// METHODS CALLS//
	IF bInit THEN
		M_Init() ; 
		bInit	:= FALSE ; 
	ELSIF CmdInit_G  THEN 
		bInit:= TRUE ;
	END_IF
	
	M_Read();
	
	M_Evaluate();
		
	M_StateManager() ; 
	M_Write();
	M_StartStop() ; 
	

	
	M_AlarmManagement();
END_METHOD

METHOD M_Init
VAR 

END_VAR
END_METHOD

METHOD M_Read
//////////////////
//  Read Modbus Variable for racks and BBMS .  
/////////////////

VAR 
	// Method local variables (reinitialized at each cycle) 

	
END_VAR
END_METHOD

METHOD M_Write
VAR_INPUT
END_VAR
VAR
	AX_ADDR 	: ARRAY[1..1] OF UINT := [1];
	AX_QTY		: ARRAY[1..1] OF BYTE := [3];
	AX_UnitID	: ARRAY[1..1] OF BYTE := [1];
END_VAR
END_METHOD

END_FUNCTION_BLOCK

// ---- 01_Equipement_Library/Batteries/FB_SystemBMS_M3.TcPOU
FUNCTION_BLOCK FB_SystemBMS_M3 EXTENDS FB_SystemBMS_Base
// Composed of Several Racks =  A System BBMS = One DC bus independant 
// 1 Racks is composed of 1 or 2 string .  >> 1 rack = one RMBS
// 1 string is composed of several modules . >> 1 string = one DC + one DC- contactor 
// Each modules is composed of several cells . 
// 17 racks  . 

VAR_INPUT PERSISTENT
		ParamIpAddress 			: STRING 	:='192.168.1.51' ; 		// IP¨Address
		ParamUnitID				: BYTE  	:= 1 ; 					// Modbus Unit ID
		ParamTcpPort			: UINT 		:= 502;					// Modbus TCP Port
		ParamReadAlarmTime		: TIME 		:= T#90S;				// Time before communication alarm
		ParamReadWarningTime	: TIME		:= T#30S;				// Time before communication warning
		ParamClockReadRack_Delay: TIME 		:= T#500ms ; 			// Delay after bbms read and before rack read
		
		ParamNbRackString		: BYTE:=1  ; // Nb of strings of module per racks . 
		ParamNbReadAtOnce		: BYTE:=10 ; // Number of racks read at the same time . 
		
END_VAR

VAR_INPUT
	//Child objects
	
END_VAR

VAR
	
	//M_EXECUTE VARIABLES//
		AX_DFV 							: ARRAY[1..13] OF FB_DetectFixedValue;	

		
		btest							: BOOL;
END_VAR

METHOD M_Evaluate : BOOL
VAR_INPUT
END_VAR
VAR
	KK: INT;
	JJ: INT ; 
	MesUmin: REAL;
	MesUdcRack: REAL;
	CalMesCCL : REAL;
	CalMesDCL : REAL;
	CalMesIdc	: REAL;
	CalMesSoC: REAL;
	CalMesSoH: REAL;
	CalMesUdc	: REAL ; 
	CalMesUdcCell : REAL ; 
	
	CalStringsInAlarm	: INT ; 
	
	
	MesGainSoCParCycle: REAL;
	CalMesUdcConnected: REAL;
	CalMesSoCConnected: REAL;

	CalProtection: UINT;
END_VAR

// GETS COM COMMANDS , OUTPUTS  , CLOCKREAD . 


AX_TrigRead[1](CLK := ClockRead);

///// CODE EMULATION ///// 

	M_Evaluate();
	
IF AX_TrigRead[1].Q THEN
MesDataExd				:= Rea.MesDataExd.MesData.; 	
 END_IF     
 


// Initialize 
CalMesIdc := 0 ; 
CalMesCCL  := 0 ; 
CalMesDCL  := 0 ;  
CalMesSoH := 0 ; 
CalMesUdcConnected := 0 ; 
CalMesSoCConnected:= 0 ;
CalMesUdc := 0 ; 
CalMesUdcCell := 0 ;
CalStringsInAlarm := 0 ;
Rea.MesDataExd.MesData.MesRackStringState := 0 ;

// Get Data from PCS 
MesDataPcs := AX_ESS[ParamEssNum].AX_PCS[ParamSystemBmsNum].MesDataExd.MesData.
// Gestion des On et Off des DC switch
TRIG_OpenDc(CLK := CmdOpenDc);
TRIG_CloseDc(CLK := CmdCloseDc);

IF TRIG_OpenDc.Q THEN
	CmdOpenDc := FALSE;
END_IF
IF TRIG_CloseDc.Q THEN
	CmdCloseDc := FALSE;
END_IF



FOR KK := 1 TO ParamNbRacks DO
	FOR JJ:= 1 TO ParamNbRackString DO 
		
  	// check if there is a protection on either string or rack level . 
		CalProtection := Rea.MesDataExd.MesData.AX_Rack[KK].AX_RACKSTRING[JJ].MesProtection1 + Rea.MesDataExd.MesData.AX_Rack[KK].AX_RACKSTRING[JJ].MesProtection2 + Rea.MesDataExd.MesData.AX_Rack[KK].AX_RACKSTRING[JJ].MesProtection3 + Rea.MesDataExd.MesData.AX_Rack[KK].AX_RACKSTRING[JJ].MesProtection4 + Rea.MesDataExd.MesData.AX_Rack[KK].MesProtection1 + Rea.MesDataExd.MesData.AX_Rack[KK].MesProtection2  ; 
		
		IF CalProtection > 0 THEN 
			CalStringsInAlarm :=  CalStringsInAlarm + 1  ;
		END_IF
		
	TRIG_OpenDcRack[KK][JJ](CLK := Rea.MesDataExd.MesData.AX_Rack[KK].AX_RACKSTRING[JJ].MesMode = 3  AND TRIG_OpenDc.Q OR CalProtection>0);		// Opens if protection alarm
	TRIG_CloseDcRack[KK][JJ](CLK := Rea.MesDataExd.MesData.AX_Rack[KK].AX_RACKSTRING[JJ].MesMode <> 3 AND TRIG_CloseDc.Q AND CalProtection=0 );	// do not close if protection alarm
	

		IF TRIG_OpenDcRack[KK][JJ].Q THEN
			Rea.MesDataExd.MesData.AX_Rack[KK].AX_RACKSTRING[1].MesMode := 2;
			//Rea.MesDataExd.MesData.AX_Rack[KK].AX_RACKSTRING[2].MesMode := 2;	
			Rea.MesDataExd.MesData.AX_Rack[KK].MesSwitchSensorStatus := 248 ;	// protections are set and fuse are ok . Dc and ac switch are opened .
			Rea.MesDataExd.MesData.AX_Rack[KK].MesDcOpenCount			:=Rea.MesDataExd.MesData.AX_Rack[KK].MesDcOpenCount +1  ;//evaluate 
				
		END_IF
		IF TRIG_CloseDcRack[KK][JJ].Q THEN
			Rea.MesDataExd.MesData.AX_Rack[KK].AX_RACKSTRING[1].MesMode := 3;
			//Rea.MesDataExd.MesData.AX_Rack[KK].AX_RACKSTRING[2].MesMode := 3;
			Rea.MesDataExd.MesData.AX_Rack[KK].MesSwitchSensorStatus := 255 ;	// protections are set and fuse are ok . Dc and ac switch are opened .
			Rea.MesDataExd.MesData.AX_Rack[KK].MesDcCloseCount			:=Rea.MesDataExd.MesData.AX_Rack[KK].MesDcCloseCount + 1			 ;//evaluate 		
		END_IF	
	END_FOR
END_FOR

NbRacksOn := 0;

FOR KK := 1 TO ParamNbRacks DO
	FOR JJ := 1 TO ParamNbRackString DO 
		IF Rea.MesDataExd.MesData.AX_Rack[KK].AX_RACKSTRING[JJ].MesMode = 3 THEN
			NbRacksOn := NbRacksOn + 1;
		END_IF
	END_FOR
END_FOR		


FOR KK := 1 TO ParamNbRacks DO
	FOR JJ := 1 TO ParamNbRackString DO 
		IF Rea.MesDataExd.MesData.AX_Rack[KK].AX_RACKSTRING[JJ].MesMode = 3 AND NbRacksOn>=1 THEN

		Rea.MesDataExd.MesData.AX_Rack[KK].AX_RACKSTRING[JJ].MesIdc := MesDataExd.MesData.cs.CalIdc / NbRacksOn;
		MesGainSoCParCycle := Rea.MesDataExd.MesData.AX_Rack[KK].AX_RACKSTRING[JJ].MesIdc*Rea.MesDataExd.MesData.AX_Rack[KK].AX_RACKSTRING[JJ].MesUdc*(ParamCycleTime_Emul/3600000.0)/(Rea.MesDataExd.MesData.AX_Rack[KK].AX_RACKSTRING[JJ].MesSoH/100.0);
		Rea.MesDataExd.MesData.AX_Rack[KK].AX_RACKSTRING[JJ].MesSoC	 	:=MIN(MAX(0, Rea.MesDataExd.MesData.AX_Rack[KK].AX_RACKSTRING[JJ].MesSoC + MesGainSoCParCycle/CstEnergyRack*100), 100); ;//evaluate 	
		Rea.MesDataExd.MesData.AX_Rack[KK].AX_RACKSTRING[JJ].MesCCL := SEL(Rea.MesDataExd.MesData.AX_Rack[KK].AX_RACKSTRING[JJ].MesSoC < 95, (100-Rea.MesDataExd.MesData.AX_Rack[KK].AX_RACKSTRING[JJ].MesSoC)*CstEnergyRack*CstMaxCrateCharge/8000, CstEnergyRack*CstMaxCrateCharge*CstNominalVoltage/Rea.MesDataExd.MesData.AX_Rack[KK].AX_RACKSTRING[JJ].MesUdc_Cell/1000);
		Rea.MesDataExd.MesData.AX_Rack[KK].AX_RACKSTRING[JJ].MesDCL := SEL(Rea.MesDataExd.MesData.AX_Rack[KK].AX_RACKSTRING[JJ].MesSoC > 5, Rea.MesDataExd.MesData.AX_Rack[KK].AX_RACKSTRING[JJ].MesSoC*CstEnergyRack*CstMaxCrateDischarge/8000, CstEnergyRack*CstMaxCrateDischarge*CstNominalVoltage/Rea.MesDataExd.MesData.AX_Rack[KK].AX_RACKSTRING[JJ].MesUdc_Cell/1000);
		Rea.MesDataExd.MesData.AX_Rack[KK].AX_RACKSTRING[JJ].MesState.1 := SEL(Rea.MesDataExd.MesData.AX_Rack[KK].AX_RACKSTRING[JJ].MesIdc <> 0 , TRUE  , FALSE )  ; 
		CalMesUdcConnected := CalMesUdcConnected + Rea.MesDataExd.MesData.AX_Rack[KK].AX_RACKSTRING[JJ].MesUdc / NbRacksOn ; 
		CalMesSoCConnected := CalMesSoCConnected  +  Rea.MesDataExd.MesData.AX_Rack[KK].AX_RACKSTRING[JJ].MesSoC / NbRacksOn ; 
		ELSE
			Rea.MesDataExd.MesData.AX_Rack[KK].AX_RACKSTRING[JJ].MesIdc := 0;
			Rea.MesDataExd.MesData.AX_Rack[KK].AX_RACKSTRING[JJ].MesCCL := 0;
			Rea.MesDataExd.MesData.AX_Rack[KK].AX_RACKSTRING[JJ].MesDCL :=0;
			Rea.MesDataExd.MesData.AX_Rack[KK].AX_RACKSTRING[JJ].MesState := 0  ; 	
		END_IF
		
		MesUmin := ParamUdcMin +(ParamUdcMax - ParamUdcMin) * Rea.MesDataExd.MesData.AX_Rack[KK].AX_RACKSTRING[JJ].MesSoC /100;
		Rea.MesDataExd.MesData.AX_Rack[KK].AX_RACKSTRING[JJ].MesUdc			:=MesUmin ;//evaluate 
		Rea.MesDataExd.MesData.AX_Rack[KK].AX_RACKSTRING[JJ].MesUdc_ModuleSum	:=MesUmin ;//evaluate 		
		Rea.MesDataExd.MesData.AX_Rack[KK].AX_RACKSTRING[JJ].MesUdc_CellSum	:=MesUmin ;//evaluate 			
		Rea.MesDataExd.MesData.AX_Rack[KK].AX_RACKSTRING[JJ].MesIdc_Avg		:=Rea.MesDataExd.MesData.AX_Rack[KK].AX_RACKSTRING[JJ].MesIdc ;//evaluate 		
			
		Rea.MesDataExd.MesData.AX_Rack[KK].AX_RACKSTRING[JJ].MesCPL		:=Rea.MesDataExd.MesData.AX_Rack[KK].AX_RACKSTRING[JJ].MesCCL * Rea.MesDataExd.MesData.AX_Rack[KK].AX_RACKSTRING[JJ].MesUdc ;//evaluate 	
		Rea.MesDataExd.MesData.AX_Rack[KK].AX_RACKSTRING[JJ].MesDPL		:=Rea.MesDataExd.MesData.AX_Rack[KK].AX_RACKSTRING[JJ].MesDCL * Rea.MesDataExd.MesData.AX_Rack[KK].AX_RACKSTRING[JJ].MesUdc ;//evaluate 

		IF Rea.MesDataExd.MesData.AX_Rack[KK].AX_RACKSTRING[JJ].MesIdc > 0 THEN 
			Rea.MesDataExd.MesData.AX_Rack[KK].AX_RACKSTRING[JJ].MesECharge := Rea.MesDataExd.MesData.AX_Rack[KK].AX_RACKSTRING[JJ].MesECharge + Rea.MesDataExd.MesData.AX_Rack[KK].AX_RACKSTRING[JJ].MesIdc*Rea.MesDataExd.MesData.AX_Rack[KK].AX_RACKSTRING[JJ].MesUdc*ParamCycleTime_Emul/3600000.0 ;
		ELSE 
			Rea.MesDataExd.MesData.AX_Rack[KK].AX_RACKSTRING[JJ].MesEDischarge := Rea.MesDataExd.MesData.AX_Rack[KK].AX_RACKSTRING[JJ].MesEDischarge - Rea.MesDataExd.MesData.AX_Rack[KK].AX_RACKSTRING[JJ].MesIdc*Rea.MesDataExd.MesData.AX_Rack[KK].AX_RACKSTRING[JJ].MesUdc*ParamCycleTime_Emul/3600000.0 ;

		END_IF

		Rea.MesDataExd.MesData.AX_Rack[KK].AX_RACKSTRING[JJ].MesUdc_Cell		:=Rea.MesDataExd.MesData.AX_Rack[KK].AX_RACKSTRING[JJ].MesUdc / 264 ;//evaluate Nb of cells per strings 
		Rea.MesDataExd.MesData.AX_Rack[KK].AX_RACKSTRING[JJ].MesUdcMax1_Cell	:=Rea.MesDataExd.MesData.AX_Rack[KK].AX_RACKSTRING[JJ].MesUdc_Cell ;//evaluate 
		Rea.MesDataExd.MesData.AX_Rack[KK].AX_RACKSTRING[JJ].MesUdcMin1_Cell:=Rea.MesDataExd.MesData.AX_Rack[KK].AX_RACKSTRING[JJ].MesUdc_Cell ;//evaluate 
		Rea.MesDataExd.MesData.AX_Rack[KK].AX_RACKSTRING[JJ].MesUdcMax2_Cell	:=Rea.MesDataExd.MesData.AX_Rack[KK].AX_RACKSTRING[JJ].MesUdc_Cell ;//evaluate 
		Rea.MesDataExd.MesData.AX_Rack[KK].AX_RACKSTRING[JJ].MesUdcMin2_Cell:=Rea.MesDataExd.MesData.AX_Rack[KK].AX_RACKSTRING[JJ].MesUdc_Cell ;//evaluate 
		
		Rea.MesDataExd.MesData.MesRackStringState			        := Rea.MesDataExd.MesData.MesRackStringState OR Rea.MesDataExd.MesData.AX_Rack[KK].AX_RACKSTRING[JJ].MesState;//evaluate 
				
		CalMesIdc := CalMesIdc +  Rea.MesDataExd.MesData.AX_Rack[KK].AX_RACKSTRING[JJ].MesIdc ;
		CalMesCCL  	:= CalMesCCL + Rea.MesDataExd.MesData.AX_Rack[KK].Ax_RACKSTRING[JJ].MesCCL; 
		CalMesDCL  	:= CalMesDCL + Rea.MesDataExd.MesData.AX_Rack[KK].Ax_RACKSTRING[JJ].MesDCL; 
		CalMesSoC 	:= CalMesSoC + Rea.MesDataExd.MesData.AX_Rack[KK].Ax_RACKSTRING[JJ].MesSoC / ParamNbRacks; 
		CalMesUdc := CalMesUdc + Rea.MesDataExd.MesData.AX_Rack[KK].AX_RACKSTRING[JJ].MesUdc / ParamNbRacks ; 
		CalMesUdcCell := CalMesUdcCell  + Rea.MesDataExd.MesData.AX_Rack[KK].AX_RACKSTRING[JJ].MesUdc_Cell / ParamNbRacks ;

	END_FOR

	Rea.MesDataExd.MesData.AX_Rack[KK].MesHeartBeat		:=WORD_TO_UINT(CalLocalTimeStruct.wSecond); ;//evaluate 

END_FOR	

Rea.MesDataExd.MesData.MesHeartBeat						:=WORD_TO_UINT(CalLocalTimeStruct.wSecond); ;//evaluate			
Rea.MesDataExd.MesData.MesNbRackConnected			        :=NbRacksOn ;//evaluate
Rea.MesDataExd.MesData.MesIdcConnected				        :=CalMesIdc ;//evaluate
Rea.MesDataExd.MesData.MesUdcConnected				        :=CalMesUdcConnected ;//evaluate
Rea.MesDataExd.MesData.MesUdcConnectedMedian		        :=CalMesUdcConnected ;//evaluate
Rea.MesDataExd.MesData.MesUdcConnectedMax			        := CalMesUdcConnected;//evaluate
Rea.MesDataExd.MesData.MesUdcConnectedMin			        := CalMesUdcConnected;//evaluate
Rea.MesDataExd.MesData.MesSoCConnected				        := CalMesSoCConnected;//evaluate average 
Rea.MesDataExd.MesData.MesSoCConnectedMedian		        := CalMesSoCConnected;//evaluate
Rea.MesDataExd.MesData.MesSoCConnectedMax			        := CalMesSoCConnected;//evaluate
Rea.MesDataExd.MesData.MesSoCConnectedMin			        := CalMesSoCConnected;//evaluate
Rea.MesDataExd.MesData.MesIdc						        := CalMesIdc;//evaluate
Rea.MesDataExd.MesData.MesUdc						        := CalMesUdc;//evaluate
Rea.MesDataExd.MesData.MesUdcMedian				        := CalMesUdc;//evaluate
Rea.MesDataExd.MesData.MesUdcMax					        := CalMesUdc;//evaluate
Rea.MesDataExd.MesData.MesUdcMin					        := CalMesUdc;//evaluate
Rea.MesDataExd.MesData.MesSoC						        := CalMesSoC;//evaluate
Rea.MesDataExd.MesData.MesSoCMedian				        := CalMesSoC;//evaluate
Rea.MesDataExd.MesData.MesSoCMax					        := CalMesSoC;//evaluate
Rea.MesDataExd.MesData.MesSoCMin					        := CalMesSoC;//evaluate
Rea.MesDataExd.MesData.MesUdc_Cell					        := CalMesUdcCell;//evaluate
Rea.MesDataExd.MesData.MesUdcMedian_Cell			        := CalMesUdcCell;//evaluate
Rea.MesDataExd.MesData.MesUdcMax_Cell				        := CalMesUdcCell;//evaluate
Rea.MesDataExd.MesData.MesUdcMin_Cell				        := CalMesUdcCell;//evaluate
Rea.MesDataExd.MesData.MesCCL						        := CalMesCCL;//evaluate
Rea.MesDataExd.MesData.MesDCL						        := CalMesDCL;//evaluate
Rea.MesDataExd.MesData.MesCPL						        := CalMesCCL *Rea.MesDataExd.MesData.MesUdc ;//evaluate
Rea.MesDataExd.MesData.MesDPL						        := CalMesDCL *Rea.MesDataExd.MesData.MesUdc;//evaluate
IF Rea.MesDataExd.MesData.MesIdc > 0 THEN 
	Rea.MesDataExd.MesData.MesECharge := Rea.MesDataExd.MesData.MesECharge + Rea.MesDataExd.MesData.MesIdc*Rea.MesDataExd.MesData.MesUdc*ParamCycleTime_Emul/3600000.0 ;
ELSE 
	Rea.MesDataExd.MesData.MesEDischarge := Rea.MesDataExd.MesData.MesEDischarge - Rea.MesDataExd.MesData.MesIdc*Rea.MesDataExd.MesData.MesUdc*ParamCycleTime_Emul/3600000.0 ;

END_IF

Rea.MesDataExd.MesData.MesWatchdog					        := AX_Cmd[3];//evaluate

Rea.MesDataExd.MesData.MesSystemMode.15				     := Rea.MesDataExd.MesData.MesIdc < - (3 * Rea.MesDataExd.MesData.MesNbRackConnected) ;//discharge 
Rea.MesDataExd.MesData.MesSystemMode.14				     := Rea.MesDataExd.MesData.MesIdc > 3  *Rea.MesDataExd.MesData.MesNbRackConnected ;//discharge 




Rea.MesDataExd.MesData.MesSystemMode.2:= SEL(CalStringsInAlarm = 0 AND Rea.MesDataExd.MesData.MesNbRackConnected =0  , FALSE ,  TRUE )  ;		// all strings can be connected 
Rea.MesDataExd.MesData.MesSystemMode.3:= NOT Rea.MesDataExd.MesData.MesSystemMode.2 AND SEL(CalStringsInAlarm < ( Rea.MesDataExd.MesData.MesNbRackTot - Rea.MesDataExd.MesData.ParamStringNbMin ) AND Rea.MesDataExd.MesData.MesNbRackConnected =0  , FALSE ,  TRUE )  ;		// Part of strings can be connected 
Rea.MesDataExd.MesData.MesSystemMode.4:= SEL(CalStringsInAlarm >= ( Rea.MesDataExd.MesData.MesNbRackTot - Rea.MesDataExd.MesData.ParamStringNbMin ) AND Rea.MesDataExd.MesData.MesNbRackConnected =0 , FALSE ,  TRUE )  ;	// 
Rea.MesDataExd.MesData.MesSystemMode.5:= SEL(CalStringsInAlarm = 0 AND Rea.MesDataExd.MesData.MesNbRackConnected >0  , FALSE ,  TRUE )  ;
Rea.MesDataExd.MesData.MesSystemMode.6:= NOT Rea.MesDataExd.MesData.MesSystemMode.5 AND SEL(CalStringsInAlarm > 0 AND Rea.MesDataExd.MesData.MesNbRackConnected =0  , FALSE ,  TRUE )  ;
END_METHOD

METHOD M_Init
VAR 
KK:  INT  ; 

	JJ: INT;
END_VAR
FOR KK := 1 TO ParamNbRacks DO
	FOR JJ := 1 TO ParamNbRackString DO 
		Rea.MesDataExd.MesData.AX_Rack[KK].AX_RACKSTRING[JJ].MesMode						:=2  ;//evaluate 				
		Rea.MesDataExd.MesData.AX_Rack[KK].AX_RACKSTRING[JJ].MesAlarm1					    :=0  ;//init 
		Rea.MesDataExd.MesData.AX_Rack[KK].AX_RACKSTRING[JJ].MesAlarm2						:=0  ;//init  	
		Rea.MesDataExd.MesData.AX_Rack[KK].AX_RACKSTRING[JJ].MesAlarm3						:=0  ;//init  	
		Rea.MesDataExd.MesData.AX_Rack[KK].AX_RACKSTRING[JJ].MesAlarm4						:=0  ;//init  	
		Rea.MesDataExd.MesData.AX_Rack[KK].AX_RACKSTRING[JJ].MesProtection1				:=0  ;//init  		
		Rea.MesDataExd.MesData.AX_Rack[KK].AX_RACKSTRING[JJ].MesProtection2				:=0  ;//init  		
		Rea.MesDataExd.MesData.AX_Rack[KK].AX_RACKSTRING[JJ].MesProtection3				:=0  ;//init  		
		Rea.MesDataExd.MesData.AX_Rack[KK].AX_RACKSTRING[JJ].MesProtection4				:=0  ;//init  		
		Rea.MesDataExd.MesData.AX_Rack[KK].AX_RACKSTRING[JJ].MesControlStatus				:=1  ;//init  	
		Rea.MesDataExd.MesData.AX_Rack[KK].AX_RACKSTRING[JJ].MesUdc						:=850  ;//evaluate 		
		Rea.MesDataExd.MesData.AX_Rack[KK].AX_RACKSTRING[JJ].MesUdc_ModuleSum				:=850  ;//evaluate	
		Rea.MesDataExd.MesData.AX_Rack[KK].AX_RACKSTRING[JJ].MesUdc_CellSum				:=850  ;//evaluate
		Rea.MesDataExd.MesData.AX_Rack[KK].AX_RACKSTRING[JJ].MesIdc						:=0  ;//evaluate	
		Rea.MesDataExd.MesData.AX_Rack[KK].AX_RACKSTRING[JJ].MesIdc_Avg					:=0  ;//evaluate	
		Rea.MesDataExd.MesData.AX_Rack[KK].AX_RACKSTRING[JJ].MesSoC	 					:=50  ;//evaluate	
		Rea.MesDataExd.MesData.AX_Rack[KK].AX_RACKSTRING[JJ].MesSoH	 					:=100  ;//evaluate	
		Rea.MesDataExd.MesData.AX_Rack[KK].AX_RACKSTRING[JJ].MesCCL						:=0  ;//evaluate	
		Rea.MesDataExd.MesData.AX_Rack[KK].AX_RACKSTRING[JJ].MesDCL						:=0  ;//evaluate	
		Rea.MesDataExd.MesData.AX_Rack[KK].AX_RACKSTRING[JJ].MesCPL						:=0  ;//evaluate	
		Rea.MesDataExd.MesData.AX_Rack[KK].AX_RACKSTRING[JJ].MesDPL						:=0  ;//evaluate	
		Rea.MesDataExd.MesData.AX_Rack[KK].AX_RACKSTRING[JJ].MesECharge					:=0  ;//evaluate	
		Rea.MesDataExd.MesData.AX_Rack[KK].AX_RACKSTRING[JJ].MesEDischarge					:=0  ;//evaluate
		Rea.MesDataExd.MesData.AX_Rack[KK].AX_RACKSTRING[JJ].MesOff_ModuleID				:=1  ;//init 		
		Rea.MesDataExd.MesData.AX_Rack[KK].AX_RACKSTRING[JJ].MesComError_ModuleID			:=1  ;//init 	
		Rea.MesDataExd.MesData.AX_Rack[KK].AX_RACKSTRING[JJ].MesUdcDiffMax_Cell			:=0  ;//init 		
		Rea.MesDataExd.MesData.AX_Rack[KK].AX_RACKSTRING[JJ].MesUdc_Cell					:=30  ;//evaluate		
		Rea.MesDataExd.MesData.AX_Rack[KK].AX_RACKSTRING[JJ].MesUdcMax1_Cell				:=30  ;//evaluate		
		Rea.MesDataExd.MesData.AX_Rack[KK].AX_RACKSTRING[JJ].MesUdcMax1_Cell_ModuleID		:=1  ;//init 	
		Rea.MesDataExd.MesData.AX_Rack[KK].AX_RACKSTRING[JJ].MesUdcMax1_Cell_CellID		:=1  ;//init 		
		Rea.MesDataExd.MesData.AX_Rack[KK].AX_RACKSTRING[JJ].MesUdcMin1_Cell				:=30  ;//evaluate		
		Rea.MesDataExd.MesData.AX_Rack[KK].AX_RACKSTRING[JJ].MesUdcMin1_Cell_ModuleID		:=1  ;//init 	
		Rea.MesDataExd.MesData.AX_Rack[KK].AX_RACKSTRING[JJ].MesUdcMin1_Cell_CellID		:=1  ;//init 		
		Rea.MesDataExd.MesData.AX_Rack[KK].AX_RACKSTRING[JJ].MesUdcMax2_Cell				:=30  ;//evaluate		
		Rea.MesDataExd.MesData.AX_Rack[KK].AX_RACKSTRING[JJ].MesUdcMax2_Cell_ModuleID		:=1  ;//init 	
		Rea.MesDataExd.MesData.AX_Rack[KK].AX_RACKSTRING[JJ].MesUdcMax2_Cell_CellID		:=1  ;//init 		
		Rea.MesDataExd.MesData.AX_Rack[KK].AX_RACKSTRING[JJ].MesUdcMin2_Cell				:=30  ;//evaluate		
		Rea.MesDataExd.MesData.AX_Rack[KK].AX_RACKSTRING[JJ].MesUdcMin2_Cell_ModuleID		:= 1 ;//init 	
		Rea.MesDataExd.MesData.AX_Rack[KK].AX_RACKSTRING[JJ].MesUdcMin2_Cell_CellID		:= 1 ;//init 		
		Rea.MesDataExd.MesData.AX_Rack[KK].AX_RACKSTRING[JJ].MesTempDiffMax_Cell			:=0  ;//init		
		Rea.MesDataExd.MesData.AX_Rack[KK].AX_RACKSTRING[JJ].MesTemp_Cell					:=25  ;// init	
		Rea.MesDataExd.MesData.AX_Rack[KK].AX_RACKSTRING[JJ].MesTempMax1_Cell				:=25  ;//init 	
		Rea.MesDataExd.MesData.AX_Rack[KK].AX_RACKSTRING[JJ].MesTempMax1_Cell_ModuleID		:=4  ;//init 	
		Rea.MesDataExd.MesData.AX_Rack[KK].AX_RACKSTRING[JJ].MesTempMax1_Cell_CellID		:=4  ;//init 		
		Rea.MesDataExd.MesData.AX_Rack[KK].AX_RACKSTRING[JJ].MesTempMin1_Cell				:=20  ;//init 	
		Rea.MesDataExd.MesData.AX_Rack[KK].AX_RACKSTRING[JJ].MesTempMin1_Cell_ModuleID		:= 1 ;//init 	
		Rea.MesDataExd.MesData.AX_Rack[KK].AX_RACKSTRING[JJ].MesTempMin1_Cell_CellID		:= 1 ;//init 		
		Rea.MesDataExd.MesData.AX_Rack[KK].AX_RACKSTRING[JJ].MesTempMax2_Cell				:=23  ;//init 	
		Rea.MesDataExd.MesData.AX_Rack[KK].AX_RACKSTRING[JJ].MesTempMax2_Cell_ModuleID		:=3  ;//init 	
		Rea.MesDataExd.MesData.AX_Rack[KK].AX_RACKSTRING[JJ].MesTempMax2_Cell_CellID		:=3  ;//init 		
		Rea.MesDataExd.MesData.AX_Rack[KK].AX_RACKSTRING[JJ].MesTempMin2_Cell				:=21  ;//init 	
		Rea.MesDataExd.MesData.AX_Rack[KK].AX_RACKSTRING[JJ].MesTempMin2_Cell_ModuleID		:=2  ;//init 	
		Rea.MesDataExd.MesData.AX_Rack[KK].AX_RACKSTRING[JJ].MesTempMin2_Cell_CellID		:=2  ;//init 		
		Rea.MesDataExd.MesData.AX_Rack[KK].AX_RACKSTRING[JJ].MesTempPCBMax					:=31  ;//init 	
		Rea.MesDataExd.MesData.AX_Rack[KK].AX_RACKSTRING[JJ].MesTempPCBMax_ModuleID		:=5  ;//init 		
		Rea.MesDataExd.MesData.AX_Rack[KK].AX_RACKSTRING[JJ].MesTempPCBMin					:=28  ;//init 	
		Rea.MesDataExd.MesData.AX_Rack[KK].AX_RACKSTRING[JJ].MesTempPCBMin_ModuleID		:=6  ;//init 		
		Rea.MesDataExd.MesData.AX_Rack[KK].AX_RACKSTRING[JJ].MesSensorStatus				:=0  ;//init 		
		Rea.MesDataExd.MesData.AX_Rack[KK].AX_RACKSTRING[JJ].MesModuleScanStatus			:=0  ;//init 		
		Rea.MesDataExd.MesData.AX_Rack[KK].AX_RACKSTRING[JJ].MesModuleBalancingStatus		:=0  ;//init 	
		Rea.MesDataExd.MesData.AX_Rack[KK].AX_RACKSTRING[JJ].MesModuleAddressStatus		:=0  ;//init 		
		Rea.MesDataExd.MesData.AX_Rack[KK].AX_RACKSTRING[JJ].MesModuleVoltageStatus		:=0  ;//init 		
		Rea.MesDataExd.MesData.AX_Rack[KK].AX_RACKSTRING[JJ].MesModuleTemperatureStatus	:=0  ;//init 		
		Rea.MesDataExd.MesData.AX_Rack[KK].AX_RACKSTRING[JJ].MesState						:=0  ;//evaluate	
		
	END_FOR
	Rea.MesDataExd.MesData.AX_Rack[KK].ParamNbStrings			:=1 ; //init 	
	Rea.MesDataExd.MesData.AX_Rack[KK].MesHeartBeat			:= 1;//evaluate 	
	Rea.MesDataExd.MesData.AX_Rack[KK].MesAlarm1				:=0 ;//init  	
	Rea.MesDataExd.MesData.AX_Rack[KK].MesAlarm2				:=0 ;//init  	
	Rea.MesDataExd.MesData.AX_Rack[KK].MesProtection1			:=0 ;//init  	
	Rea.MesDataExd.MesData.AX_Rack[KK].MesProtection2			:=0 ;//init  	
	Rea.MesDataExd.MesData.AX_Rack[KK].MesSwitchControlStatus	:=0 ;//init  	
	Rea.MesDataExd.MesData.AX_Rack[KK].MesSwitchSensorStatus	:=0 ;//evaluate  	
	Rea.MesDataExd.MesData.AX_Rack[KK].MesUSwtchGrPackPlus		:=48 ;//init  	
	Rea.MesDataExd.MesData.AX_Rack[KK].MesTempPCB				:=25.5 ;//init  
	Rea.MesDataExd.MesData.AX_Rack[KK].MesIdcFaultLvl			:=79 ;//init  
	Rea.MesDataExd.MesData.AX_Rack[KK].MesDcOpenCount			:=0 ;//evaluate 
	Rea.MesDataExd.MesData.AX_Rack[KK].MesDcCloseCount			:=0 ;//evaluate 
	
		
END_FOR	
Rea.MesDataExd.MesData.MesHeartBeat						:=1 ;//evaluate			
Rea.MesDataExd.MesData.MesNbRackConnected			        :=17 ;//evaluate
Rea.MesDataExd.MesData.MesNbRackTot				        :=17 ;//evaluate 
Rea.MesDataExd.MesData.MesIdcConnected				        :=0 ;//evaluate
Rea.MesDataExd.MesData.MesUdcConnected				        :=850 ;//evaluate
Rea.MesDataExd.MesData.MesUdcConnectedMedian		        :=850 ;//evaluate
Rea.MesDataExd.MesData.MesUdcConnectedMax			        := 850;//evaluate
Rea.MesDataExd.MesData.MesUdcConnectedMin			        := 850;//evaluate
Rea.MesDataExd.MesData.MesSoCConnected				        := 50;//evaluate
Rea.MesDataExd.MesData.MesSoCConnectedMedian		        := 50;//evaluate
Rea.MesDataExd.MesData.MesSoCConnectedMax			        := 50;//evaluate
Rea.MesDataExd.MesData.MesSoCConnectedMin			        := 50;//evaluate
Rea.MesDataExd.MesData.MesIdc						        := 0;//evaluate
Rea.MesDataExd.MesData.MesUdc						        := 850;//evaluate
Rea.MesDataExd.MesData.MesUdcMedian				        := 850;//evaluate
Rea.MesDataExd.MesData.MesUdcMax					        := 850;//evaluate
Rea.MesDataExd.MesData.MesUdcMin					        := 850;//evaluate
Rea.MesDataExd.MesData.MesSoC						        := 50;//evaluate
Rea.MesDataExd.MesData.MesSoCMedian				        := 50;//evaluate
Rea.MesDataExd.MesData.MesSoCMax					        := 50;//evaluate
Rea.MesDataExd.MesData.MesSoCMin					        := 50;//evaluate
Rea.MesDataExd.MesData.MesSoH						        := 100;//init
Rea.MesDataExd.MesData.MesSoHMedian				        := 100;//init 
Rea.MesDataExd.MesData.MesSoHMax					        := 100;//init 
Rea.MesDataExd.MesData.MesSoHMin					        := 100;//init 
Rea.MesDataExd.MesData.MesUdc_Cell					        := 30;//evaluate
Rea.MesDataExd.MesData.MesUdcMedian_Cell			        := 30;//evaluate
Rea.MesDataExd.MesData.MesUdcMax_Cell				        := 30;//evaluate
Rea.MesDataExd.MesData.MesUdcMax_Cell_RackID		        := 30;//init 
Rea.MesDataExd.MesData.MesUdcMin_Cell				        := 30;//evaluate
Rea.MesDataExd.MesData.MesUdcMin_Cell_RackID		        := 1;//init 
Rea.MesDataExd.MesData.MesUdcDiffMax_Cell			        :=0 ;//init
Rea.MesDataExd.MesData.MesUdcDiffMax_Cell_RackID	        := 1;//init 
Rea.MesDataExd.MesData.MesTmp_Cell					        := 25;//init 
Rea.MesDataExd.MesData.MesTmpMedian_Cell			        := 25;//init 
Rea.MesDataExd.MesData.MesTmpMax_Cell				        := 25;//init 
Rea.MesDataExd.MesData.MesTmpMax_Cell_RackID		        := 3;//init 
Rea.MesDataExd.MesData.MesTmpMin_Cell				        := 25;//init 
Rea.MesDataExd.MesData.MesTmpMin_Cell_RackID		        := 4;//init 
Rea.MesDataExd.MesData.MesTmpDiffMax_Cell			        := 0;//init 
Rea.MesDataExd.MesData.MesTmpDiffMax_Cell_RackID	        := 3;//init 
Rea.MesDataExd.MesData.MesCCL						        := 0;//evaluate
Rea.MesDataExd.MesData.MesDCL						        := 0;//evaluate
Rea.MesDataExd.MesData.MesCPL						        := 0;//evaluate
Rea.MesDataExd.MesData.MesDPL						        := 0;//evaluate
Rea.MesDataExd.MesData.MesECharge					        := 0;//evaluate
Rea.MesDataExd.MesData.MesEDischarge				        := 0;//evaluate
Rea.MesDataExd.MesData.MesWatchdog					        := 0;//evaluate
Rea.MesDataExd.MesData.MesUdc_PartialOp			        := 850;//evaluate
Rea.MesDataExd.MesData.MesUdc_PartialOp_RackID		        := 8;//init 
Rea.MesDataExd.MesData.MesUdc_PartialOp_StringID	        := 3;//init 
Rea.MesDataExd.MesData.MesSystemCommandStatus		        := 0;//init 
Rea.MesDataExd.MesData.MesSystemMode				        := 0;//evaluate 
Rea.MesDataExd.MesData.MesSystemMode2				        := 0;//evaluate 
Rea.MesDataExd.MesData.MesAlarm1					        := 0;//init 
Rea.MesDataExd.MesData.MesAlarm2					        := 0;//init 
Rea.MesDataExd.MesData.MesRackAlarm1				        := 0;//init
Rea.MesDataExd.MesData.MesRackAlarm2				        := 0;//init
Rea.MesDataExd.MesData.MesRackProtection1			        := 0;//init
Rea.MesDataExd.MesData.MesRackProtection2			        := 0;//init
Rea.MesDataExd.MesData.MesRackStringAlarm1			        := 0;//init
Rea.MesDataExd.MesData.MesRackStringAlarm2			        := 0;//init
Rea.MesDataExd.MesData.MesRackStringAlarm3			        := 0;//init
Rea.MesDataExd.MesData.MesRackStringAlarm4			        := 0;//init
Rea.MesDataExd.MesData.MesRackStringProtection1	        := 0;//init
Rea.MesDataExd.MesData.MesRackStringProtection2	        := 0;//init
Rea.MesDataExd.MesData.MesRackStringProtection3	        := 0;//init
Rea.MesDataExd.MesData.MesRackStringProtection4	        := 0;//init
Rea.MesDataExd.MesData.MesDiStatus					        := 0;//init
Rea.MesDataExd.MesData.MesDoStatus					        := 0;//init
Rea.MesDataExd.MesData.MesSystemConfig1			        := 0;//init
Rea.MesDataExd.MesData.MesSystemConfig2			        := 0;//init
Rea.MesDataExd.MesData.MesRackStringState			        := 0;//evaluate 
Rea.MesDataExd.MesData.ParamNbRacks				        := 17;//init
Rea.MesDataExd.MesData.ParamNbModule				        := 25;//init
Rea.MesDataExd.MesData.ParamStringNbMin			        := 10;//init
Rea.MesDataExd.MesData.ParamUdiff					        := 5;//init


SUPER^.M_Init() ;
END_METHOD

METHOD M_Read
//////////////////
//  Read CAN 2.0B Variables for racks and BBMS .  
/////////////////

VAR 
	// Method local variables (reinitialized at each cycle) 
	MW 	: FB_MergeWordsToDint ; 

	AX_Addr		: ARRAY[1..2] OF UINT := [16#00	,  16#3E8];
	AX_Qty		: ARRAY[1..3] OF UINT := [	112		, 35	,97	];
	LL			: INT;
	KK			: BYTE;
	CalRackNb	: INT;
	JJ			: BYTE;

END_VAR
// System BMS 
IF MesCP_Read  THEN	

	ModbusRead
	(
		pDestAddr 		:= ADR(MesBlock1_Temp),		sIPAddr 		:= ParamIpAddress,			tTimeout 		:= ParamTimeout,
		nTcpPort 		:= ParamTcpPort,				nQuantity 		:= AX_Qty[1],				nMBAddr 		:= AX_Addr[1],				
		cbLength 		:= SIZEOF(MesBlock1_Temp),	nUnitID 		:= ParamUnitID,				ClockRead 		:= Clockread AND  MesCP_Read,
		Reset 			:= IN_CmdReset_L,					ModbusReadAlarm => MesModbusReadAlarm,	ErrorId 		=> MesModbusReadAlarmID
	);



MesDataExd.MesData.MesHeartBeat:=MesBlock1_Temp[0];
MesDataExd.MesData.MesNbRackConnected:=MesBlock1_Temp[1];
MesDataExd.MesData.MesNbRackTot:=MesBlock1_Temp[2];
	MW(WORD_STRONG:= MesBlock1_Temp[ 3], SIGNED:=TRUE, FIX:=0 , SIZE:=1, VAR_OUT := MesDataExd.MesData.MesIdcConnected);
	MW(WORD_STRONG:= MesBlock1_Temp[ 4], SIGNED:=FALSE, FIX:=1 , SIZE:=1, VAR_OUT := MesDataExd.MesData.MesUdcConnected);
	MW(WORD_STRONG:= MesBlock1_Temp[ 5], SIGNED:=FALSE, FIX:=1 , SIZE:=1, VAR_OUT := MesDataExd.MesData.MesUdcConnectedMedian);
	MW(WORD_STRONG:= MesBlock1_Temp[ 6], SIGNED:=FALSE, FIX:=1 , SIZE:=1, VAR_OUT := MesDataExd.MesData.MesUdcConnectedMax);
	MW(WORD_STRONG:= MesBlock1_Temp[ 7], SIGNED:=FALSE, FIX:=1 , SIZE:=1, VAR_OUT := MesDataExd.MesData.MesUdcConnectedMin);
	MW(WORD_STRONG:= MesBlock1_Temp[ 8], SIGNED:=FALSE, FIX:=1 , SIZE:=1, VAR_OUT := MesDataExd.MesData.MesSoCConnected);
	MW(WORD_STRONG:= MesBlock1_Temp[ 9], SIGNED:=FALSE, FIX:=1 , SIZE:=1, VAR_OUT := MesDataExd.MesData.MesSoCConnectedMedian);
	MW(WORD_STRONG:= MesBlock1_Temp[ 10], SIGNED:=FALSE, FIX:=1 , SIZE:=1, VAR_OUT := MesDataExd.MesData.MesSoCConnectedMax);
	MW(WORD_STRONG:= MesBlock1_Temp[ 11], SIGNED:=FALSE, FIX:=1 , SIZE:=1, VAR_OUT := MesDataExd.MesData.MesSoCConnectedMin);
	MW(WORD_STRONG:= MesBlock1_Temp[ 12], SIGNED:=TRUE, FIX:=0 , SIZE:=1, VAR_OUT := MesDataExd.MesData.MesIdc);
	MW(WORD_STRONG:= MesBlock1_Temp[ 13], SIGNED:=FALSE, FIX:=1 , SIZE:=1, VAR_OUT := MesDataExd.MesData.MesUdc);
	MW(WORD_STRONG:= MesBlock1_Temp[ 14], SIGNED:=FALSE, FIX:=1 , SIZE:=1, VAR_OUT := MesDataExd.MesData.MesUdcMedian);
	MW(WORD_STRONG:= MesBlock1_Temp[ 15], SIGNED:=FALSE, FIX:=1 , SIZE:=1, VAR_OUT := MesDataExd.MesData.MesUdcMax);
	MW(WORD_STRONG:= MesBlock1_Temp[ 16], SIGNED:=FALSE, FIX:=1 , SIZE:=1, VAR_OUT := MesDataExd.MesData.MesUdcMin);
	MW(WORD_STRONG:= MesBlock1_Temp[ 17], SIGNED:=FALSE, FIX:=1 , SIZE:=1, VAR_OUT := MesDataExd.MesData.MesSoC);
	MW(WORD_STRONG:= MesBlock1_Temp[ 18], SIGNED:=FALSE, FIX:=1 , SIZE:=1, VAR_OUT := MesDataExd.MesData.MesSoCMedian);
	MW(WORD_STRONG:= MesBlock1_Temp[ 19], SIGNED:=FALSE, FIX:=1 , SIZE:=1, VAR_OUT := MesDataExd.MesData.MesSoCMax);
	MW(WORD_STRONG:= MesBlock1_Temp[ 20], SIGNED:=FALSE, FIX:=1 , SIZE:=1, VAR_OUT := MesDataExd.MesData.MesSoCMin);
	MW(WORD_STRONG:= MesBlock1_Temp[ 21], SIGNED:=FALSE, FIX:=1 , SIZE:=1, VAR_OUT := MesDataExd.MesData.MesSoH);
	MW(WORD_STRONG:= MesBlock1_Temp[ 22], SIGNED:=FALSE, FIX:=1 , SIZE:=1, VAR_OUT := MesDataExd.MesData.MesSoHMedian);
	MW(WORD_STRONG:= MesBlock1_Temp[ 23], SIGNED:=FALSE, FIX:=1 , SIZE:=1, VAR_OUT := MesDataExd.MesData.MesSoHMax);
	MW(WORD_STRONG:= MesBlock1_Temp[ 24], SIGNED:=FALSE, FIX:=1 , SIZE:=1, VAR_OUT := MesDataExd.MesData.MesSoHMin);
	MW(WORD_STRONG:= MesBlock1_Temp[ 25], SIGNED:=FALSE, FIX:=3 , SIZE:=1, VAR_OUT := MesDataExd.MesData.MesUdc_Cell);
	MW(WORD_STRONG:= MesBlock1_Temp[ 26], SIGNED:=FALSE, FIX:=3 , SIZE:=1, VAR_OUT := MesDataExd.MesData.MesUdcMedian_Cell);
	MW(WORD_STRONG:= MesBlock1_Temp[ 27], SIGNED:=FALSE, FIX:=3 , SIZE:=1, VAR_OUT := MesDataExd.MesData.MesUdcMax_Cell);
MesDataExd.MesData.MesUdcMax_Cell_RackID:=MesBlock1_Temp[28];
	MW(WORD_STRONG:= MesBlock1_Temp[ 29], SIGNED:=FALSE, FIX:=3 , SIZE:=1, VAR_OUT := MesDataExd.MesData.MesUdcMin_Cell);
MesDataExd.MesData.MesUdcMin_Cell_RackID:=MesBlock1_Temp[30];
	MW(WORD_STRONG:= MesBlock1_Temp[ 31], SIGNED:=FALSE, FIX:=3 , SIZE:=1, VAR_OUT := MesDataExd.MesData.MesUdcDiffMax_Cell);
MesDataExd.MesData.MesUdcDiffMax_Cell_RackID:=MesBlock1_Temp[32];
	MW(WORD_STRONG:= MesBlock1_Temp[ 33], SIGNED:=TRUE, FIX:=2 , SIZE:=1, VAR_OUT := MesDataExd.MesData.MesTmp_Cell);
	MW(WORD_STRONG:= MesBlock1_Temp[ 34], SIGNED:=TRUE, FIX:=2 , SIZE:=1, VAR_OUT := MesDataExd.MesData.MesTmpMedian_Cell);
	MW(WORD_STRONG:= MesBlock1_Temp[ 35], SIGNED:=TRUE, FIX:=2 , SIZE:=1, VAR_OUT := MesDataExd.MesData.MesTmpMax_Cell);
MesDataExd.MesData.MesTmpMax_Cell_RackID:=MesBlock1_Temp[36];
	MW(WORD_STRONG:= MesBlock1_Temp[ 37], SIGNED:=TRUE, FIX:=2 , SIZE:=1, VAR_OUT := MesDataExd.MesData.MesTmpMin_Cell);
MesDataExd.MesData.MesTmpMin_Cell_RackID:=MesBlock1_Temp[38];
	MW(WORD_STRONG:= MesBlock1_Temp[ 39], SIGNED:=FALSE, FIX:=2 , SIZE:=1, VAR_OUT := MesDataExd.MesData.MesTmpDiffMax_Cell);
MesDataExd.MesData.MesTmpDiffMax_Cell_RackID:=MesBlock1_Temp[40];
	MW(WORD_STRONG:= MesBlock1_Temp[ 41], Word_WEAK:= MesBlock1_Temp[42], SIGNED:=FALSE, FIX:=1 , SIZE:=2, VAR_OUT := MesDataExd.MesData.MesCCL);
	MW(WORD_STRONG:= MesBlock1_Temp[ 43], Word_WEAK:= MesBlock1_Temp[44], SIGNED:=FALSE, FIX:=1 , SIZE:=2, VAR_OUT := MesDataExd.MesData.MesDCL);
	MW(WORD_STRONG:= MesBlock1_Temp[ 45], Word_WEAK:= MesBlock1_Temp[46], SIGNED:=FALSE, FIX:=2 , SIZE:=2, VAR_OUT := MesDataExd.MesData.MesCPL);
	MW(WORD_STRONG:= MesBlock1_Temp[ 47], Word_WEAK:= MesBlock1_Temp[48], SIGNED:=FALSE, FIX:=2 , SIZE:=2, VAR_OUT := MesDataExd.MesData.MesDPL);
	
MesDataExd.MesData.MesECharge :=  LREAL_TO_REAL(LWORD_TO_LREAL(SHL(WORD_TO_LWORD(MesBlock1_Temp[ 49]),48) OR SHL(WORD_TO_LWORD(MesBlock1_Temp[ 50]),32) OR SHL(WORD_TO_LWORD(MesBlock1_Temp[ 51]),16) OR WORD_TO_LWORD(MesBlock1_Temp[ 52]))/ EXPT(10,3) ); 
MesDataExd.MesData.MesEDischarge :=   LREAL_TO_REAL(LWORD_TO_LREAL(SHL(WORD_TO_LWORD(MesBlock1_Temp[ 53]),48) OR SHL(WORD_TO_LWORD(MesBlock1_Temp[ 54]),32) OR SHL(WORD_TO_LWORD(MesBlock1_Temp[ 55]),16) OR WORD_TO_LWORD(MesBlock1_Temp[ 56]))/ EXPT(10,3)) ; 
	
MesDataExd.MesData.MesWatchdog:=MesBlock1_Temp[57];
	MW(WORD_STRONG:= MesBlock1_Temp[ 58], SIGNED:=FALSE, FIX:=1 , SIZE:=1, VAR_OUT := MesDataExd.MesData.MesUdc_PartialOp);
MesDataExd.MesData.MesUdc_PartialOp_RackID:=MesBlock1_Temp[59];
MesDataExd.MesData.MesUdc_PartialOp_StringID:=MesBlock1_Temp[60];
MesDataExd.MesData.MesSystemCommandStatus:=MesBlock1_Temp[71];
MesDataExd.MesData.MesSystemMode:=MesBlock1_Temp[72];
MesDataExd.MesData.MesSystemMode2:=MesBlock1_Temp[73];
MesDataExd.MesData.MesAlarm1:=MesBlock1_Temp[74];
MesDataExd.MesData.MesAlarm2:=MesBlock1_Temp[75];
MesDataExd.MesData.MesRackAlarm1:=MesBlock1_Temp[76];
MesDataExd.MesData.MesRackAlarm2:=MesBlock1_Temp[77];
MesDataExd.MesData.MesRackProtection1:=MesBlock1_Temp[78];
MesDataExd.MesData.MesRackProtection2:=MesBlock1_Temp[79];
MesDataExd.MesData.MesRackStringAlarm1:=MesBlock1_Temp[80];
MesDataExd.MesData.MesRackStringAlarm2:=MesBlock1_Temp[81];
MesDataExd.MesData.MesRackStringAlarm3:=MesBlock1_Temp[82];
MesDataExd.MesData.MesRackStringAlarm4:=MesBlock1_Temp[83];
MesDataExd.MesData.MesRackStringProtection1:=MesBlock1_Temp[84];
MesDataExd.MesData.MesRackStringProtection2:=MesBlock1_Temp[85];
MesDataExd.MesData.MesRackStringProtection3:=MesBlock1_Temp[86];
MesDataExd.MesData.MesRackStringProtection4:=MesBlock1_Temp[87];
MesDataExd.MesData.MesDiStatus:=MesBlock1_Temp[88];
MesDataExd.MesData.MesDoStatus:=MesBlock1_Temp[89];
MesDataExd.MesData.MesSystemConfig1:=MesBlock1_Temp[90];
MesDataExd.MesData.MesSystemConfig2:=MesBlock1_Temp[91];
MesDataExd.MesData.MesRackStringState:=MesBlock1_Temp[92];
MesDataExd.MesData.ParamNbRacks:=MesBlock1_Temp[105];
MesDataExd.MesData.ParamNbModule:=MesBlock1_Temp[106];
MesDataExd.MesData.ParamStringNbMin:=MesBlock1_Temp[107];
	MW(WORD_STRONG:= MesBlock1_Temp[ 108], SIGNED:=FALSE, FIX:=0 , SIZE:=1, VAR_OUT := MesDataExd.MesData.ParamUdiff);

END_IF
// RACKS 

// READ TCU DATA 
CTU_ClockRead(CU:=ClockRead , PV:= REAL_TO_WORD(ParamNbRacks/(ParamNbReadAtOnce))+1 ) ; 
CTU_ClockRead(RESET:= CTU_ClockRead.Q ) ; 
LL:= (CTU_ClockRead.CV)  ; // At every Clock Read , we read 10 new racks We reset once all trackers have been read.  


TON_ClockRead(IN:= ClockRead , PT:= ParamClockReadRack_Delay  ) ; // Allow to leave 200ms between the system data read and the racks reading . 

//RACK 
FOR KK:= 1 TO ParamNbReadAtOnce DO 
	
	CalRackNb := LL*ParamNbReadAtOnce+KK; 	
	IF CalRackNb > ParamNbRacks THEN 
		EXIT ; 
	END_IF	
	
	IF MesCP_Read THEN
		ModbusReadrack[(ParamNbRackString+1)*(KK-1)+1]
			(
			pDestAddr 		:= ADR(MesBlock2_Temp[(ParamNbRackString+1)*(KK-1)+1]),		sIPAddr 		:= ParamIpAddress,			tTimeout 		:= ParamTimeout,
			nTcpPort 		:= ParamTcpPort,				nQuantity 		:= AX_Qty[2],				nMBAddr 		:= AX_Addr[2] + (CalRackNb-1)*360,				
			cbLength 		:= SIZEOF(MesBlock2_Temp[(ParamNbRackString+1)*(KK-1)+1]),	nUnitID 		:= ParamUnitID,				ClockRead 		:= TON_ClockRead.Q AND MesCP_Read,
			Reset 			:= IN_CmdReset_L,					ModbusReadAlarm => MesModbusReadAlarm2[(ParamNbRackString+1)*(KK-1)+1],	ErrorId 		=> MesModbusReadAlarmID2[(ParamNbRackString+1)*(KK-1)+1]
		);
	

	// DATA
		IF ModbusReadrack[(ParamNbRackString+1)*(KK-1)+1].OUT_Completed THEN 
		MesDataExd.MesData.AX_Rack[CalRackNb].ParamNbStrings:=MesBlock2_Temp[(ParamNbRackString+1)*(KK-1)+1][0];
		MesDataExd.MesData.AX_Rack[CalRackNb].MesHeartBeat:=MesBlock2_Temp[(ParamNbRackString+1)*(KK-1)+1][1];
		MesDataExd.MesData.AX_Rack[CalRackNb].MesAlarm1:=MesBlock2_Temp[(ParamNbRackString+1)*(KK-1)+1][2];
		MesDataExd.MesData.AX_Rack[CalRackNb].MesAlarm2:=MesBlock2_Temp[(ParamNbRackString+1)*(KK-1)+1][3];
		MesDataExd.MesData.AX_Rack[CalRackNb].MesProtection1:=MesBlock2_Temp[(ParamNbRackString+1)*(KK-1)+1][4];
		MesDataExd.MesData.AX_Rack[CalRackNb].MesProtection2:=MesBlock2_Temp[(ParamNbRackString+1)*(KK-1)+1][5];
		MesDataExd.MesData.AX_Rack[CalRackNb].MesState_SwitchControl:=MesBlock2_Temp[(ParamNbRackString+1)*(KK-1)+1][6];
		MesDataExd.MesData.AX_Rack[CalRackNb].MesState_SwitchSensor:=MesBlock2_Temp[(ParamNbRackString+1)*(KK-1)+1][7];
			MW(WORD_STRONG:= MesBlock2_Temp[(ParamNbRackString+1)*(KK-1)+1][ 10], 	SIGNED:=FALSE, FIX:=1 , SIZE:=1, VAR_OUT := MesDataExd.MesData.AX_Rack[CalRackNb].MesUPackPlus_SwtchGr);
			MW(WORD_STRONG:= MesBlock2_Temp[(ParamNbRackString+1)*(KK-1)+1][ 12], 	SIGNED:=TRUE, FIX:=0 , SIZE:=1, VAR_OUT := MesDataExd.MesData.AX_Rack[CalRackNb].MesTempPCB);
		MesDataExd.MesData.AX_Rack[CalRackNb].MesIdcFaultLvl:=MesBlock2_Temp[(ParamNbRackString+1)*(KK-1)+1][23];
		MesDataExd.MesData.AX_Rack[CalRackNb].MesDcOpenCount:=MesBlock2_Temp[(ParamNbRackString+1)*(KK-1)+1][24];
		MesDataExd.MesData.AX_Rack[CalRackNb].MesDcCloseCount:=MesBlock2_Temp[(ParamNbRackString+1)*(KK-1)+1][25];
		END_IF
	END_IF
	// RACK STRING 
	FOR JJ:= 1 TO ParamNbRackString DO 
		IF MesCP_Read THEN	
			ModbusReadrack[(ParamNbRackString+1)*(KK-1)+JJ+1]
				(
				pDestAddr 		:= ADR(MesBlock2_Temp[(ParamNbRackString+1)*(KK-1)+JJ+1]),		sIPAddr 		:= ParamIpAddress,			tTimeout 		:= ParamTimeout,
				nTcpPort 		:= ParamTcpPort,				nQuantity 		:= AX_Qty[3],				nMBAddr 		:= AX_Addr[2] + (CalRackNb-1)*360 + JJ*120,				
				cbLength 		:= SIZEOF(MesBlock2_Temp[(ParamNbRackString+1)*(KK-1)+JJ+1]),	nUnitID 		:= ParamUnitID,				ClockRead 		:= TON_ClockRead.Q AND MesCP_Read,
				Reset 			:= IN_CmdReset_L,					ModbusReadAlarm => MesModbusReadAlarm2[(ParamNbRackString+1)*(KK-1)+JJ+1],	ErrorId 		=> MesModbusReadAlarmID2[(ParamNbRackString+1)*(KK-1)+JJ+1]
			);

		//DATA
			IF ModbusReadrack[(ParamNbRackString+1)*(KK-1)+JJ+1].OUT_Completed THEN 
			MesDataExd.MesData.AX_RACK[CalrackNb].AX_RACKSTRING[JJ].MesMode:=MesBlock2_Temp[(ParamNbRackString+1)*(KK-1)+JJ+1][0];
			MesDataExd.MesData.AX_RACK[CalrackNb].AX_RACKSTRING[JJ].MesAlarm1:=MesBlock2_Temp[(ParamNbRackString+1)*(KK-1)+JJ+1][2];
			MesDataExd.MesData.AX_RACK[CalrackNb].AX_RACKSTRING[JJ].MesAlarm2:=MesBlock2_Temp[(ParamNbRackString+1)*(KK-1)+JJ+1][3];
			MesDataExd.MesData.AX_RACK[CalrackNb].AX_RACKSTRING[JJ].MesAlarm3:=MesBlock2_Temp[(ParamNbRackString+1)*(KK-1)+JJ+1][4];
			MesDataExd.MesData.AX_RACK[CalrackNb].AX_RACKSTRING[JJ].MesAlarm4:=MesBlock2_Temp[(ParamNbRackString+1)*(KK-1)+JJ+1][5];
			MesDataExd.MesData.AX_RACK[CalrackNb].AX_RACKSTRING[JJ].MesProtection1:=MesBlock2_Temp[(ParamNbRackString+1)*(KK-1)+JJ+1][6];
			MesDataExd.MesData.AX_RACK[CalrackNb].AX_RACKSTRING[JJ].MesProtection2:=MesBlock2_Temp[(ParamNbRackString+1)*(KK-1)+JJ+1][7];
			MesDataExd.MesData.AX_RACK[CalrackNb].AX_RACKSTRING[JJ].MesProtection3:=MesBlock2_Temp[(ParamNbRackString+1)*(KK-1)+JJ+1][8];
			MesDataExd.MesData.AX_RACK[CalrackNb].AX_RACKSTRING[JJ].MesProtection4:=MesBlock2_Temp[(ParamNbRackString+1)*(KK-1)+JJ+1][9];
			MesDataExd.MesData.AX_RACK[CalrackNb].AX_RACKSTRING[JJ].MesControlStatus:=MesBlock2_Temp[(ParamNbRackString+1)*(KK-1)+JJ+1][10];
				MW(WORD_STRONG:= MesBlock2_Temp[(ParamNbRackString+1)*(KK-1)+JJ+1][ 13], SIGNED:=FALSE, FIX:=1 , SIZE:=1, VAR_OUT := MesDataExd.MesData.AX_RACK[CalrackNb].AX_RACKSTRING[JJ].MesUdc);
				MW(WORD_STRONG:= MesBlock2_Temp[(ParamNbRackString+1)*(KK-1)+JJ+1][ 14], SIGNED:=FALSE, FIX:=1 , SIZE:=1, VAR_OUT := MesDataExd.MesData.AX_RACK[CalrackNb].AX_RACKSTRING[JJ].MesUdc_ModuleSum);
				MW(WORD_STRONG:= MesBlock2_Temp[(ParamNbRackString+1)*(KK-1)+JJ+1][ 15], SIGNED:=FALSE, FIX:=1 , SIZE:=1, VAR_OUT := MesDataExd.MesData.AX_RACK[CalrackNb].AX_RACKSTRING[JJ].MesUdc_CellSum);
				MW(WORD_STRONG:= MesBlock2_Temp[(ParamNbRackString+1)*(KK-1)+JJ+1][ 16], SIGNED:=TRUE, FIX:=1 , SIZE:=1, VAR_OUT := MesDataExd.MesData.AX_RACK[CalrackNb].AX_RACKSTRING[JJ].MesIdc);
				MW(WORD_STRONG:= MesBlock2_Temp[(ParamNbRackString+1)*(KK-1)+JJ+1][ 17], SIGNED:=TRUE, FIX:=1 , SIZE:=1, VAR_OUT := MesDataExd.MesData.AX_RACK[CalrackNb].AX_RACKSTRING[JJ].MesIdc_Avg);
				MW(WORD_STRONG:= MesBlock2_Temp[(ParamNbRackString+1)*(KK-1)+JJ+1][ 18], SIGNED:=FALSE, FIX:=1 , SIZE:=1, VAR_OUT := MesDataExd.MesData.AX_RACK[CalrackNb].AX_RACKSTRING[JJ].MesSoC);
				MW(WORD_STRONG:= MesBlock2_Temp[(ParamNbRackString+1)*(KK-1)+JJ+1][ 19], SIGNED:=FALSE, FIX:=1 , SIZE:=1, VAR_OUT := MesDataExd.MesData.AX_RACK[CalrackNb].AX_RACKSTRING[JJ].MesSoH);
				MW(WORD_STRONG:= MesBlock2_Temp[(ParamNbRackString+1)*(KK-1)+JJ+1][ 20], SIGNED:=FALSE, FIX:=1 , SIZE:=1, VAR_OUT := MesDataExd.MesData.AX_RACK[CalrackNb].AX_RACKSTRING[JJ].MesCCL);
				MW(WORD_STRONG:= MesBlock2_Temp[(ParamNbRackString+1)*(KK-1)+JJ+1][ 21], SIGNED:=FALSE, FIX:=1 , SIZE:=1, VAR_OUT := MesDataExd.MesData.AX_RACK[CalrackNb].AX_RACKSTRING[JJ].MesDCL);
				MW(WORD_STRONG:= MesBlock2_Temp[(ParamNbRackString+1)*(KK-1)+JJ+1][ 22], SIGNED:=FALSE, FIX:=2 , SIZE:=1, VAR_OUT := MesDataExd.MesData.AX_RACK[CalrackNb].AX_RACKSTRING[JJ].MesCPL);
				MW(WORD_STRONG:= MesBlock2_Temp[(ParamNbRackString+1)*(KK-1)+JJ+1][ 23], SIGNED:=FALSE, FIX:=2 , SIZE:=1, VAR_OUT := MesDataExd.MesData.AX_RACK[CalrackNb].AX_RACKSTRING[JJ].MesDPL);
				
			MesDataExd.MesData.AX_RACK[CalrackNb].AX_RACKSTRING[JJ].MesECharge := LREAL_TO_REAL(LWORD_TO_LREAL(SHL(WORD_TO_LWORD(MesBlock2_Temp[(ParamNbRackString+1)*(KK-1)+JJ+1][ 24]),48) OR SHL(WORD_TO_LWORD(MesBlock2_Temp[(ParamNbRackString+1)*(KK-1)+JJ+1][ 25]),32) OR SHL(WORD_TO_LWORD(MesBlock2_Temp[(ParamNbRackString+1)*(KK-1)+JJ+1][ 26]),16) OR WORD_TO_LWORD(MesBlock2_Temp[(ParamNbRackString+1)*(KK-1)+JJ+1][ 27]))/ EXPT(10,3) ); 
				
			MesDataExd.MesData.AX_RACK[CalrackNb].AX_RACKSTRING[JJ].MesEDischarge := LREAL_TO_REAL(LWORD_TO_LREAL(SHL(WORD_TO_LWORD(MesBlock2_Temp[(ParamNbRackString+1)*(KK-1)+JJ+1][ 28]),48) OR SHL(WORD_TO_LWORD(MesBlock2_Temp[(ParamNbRackString+1)*(KK-1)+JJ+1][ 29]),32) OR SHL(WORD_TO_LWORD(MesBlock2_Temp[(ParamNbRackString+1)*(KK-1)+JJ+1][ 30]),16) OR WORD_TO_LWORD(MesBlock2_Temp[(ParamNbRackString+1)*(KK-1)+JJ+1][ 31]))/ EXPT(10,3) ); 
				
			MesDataExd.MesData.AX_RACK[CalrackNb].AX_RACKSTRING[JJ].MesOff_ModuleID:=MesBlock2_Temp[(ParamNbRackString+1)*(KK-1)+JJ+1][36];
			MesDataExd.MesData.AX_RACK[CalrackNb].AX_RACKSTRING[JJ].MesComError_ModuleID:=MesBlock2_Temp[(ParamNbRackString+1)*(KK-1)+JJ+1][37];
				MW(WORD_STRONG:= MesBlock2_Temp[(ParamNbRackString+1)*(KK-1)+JJ+1][ 38], SIGNED:=FALSE, FIX:=3 , SIZE:=1, VAR_OUT := MesDataExd.MesData.AX_RACK[CalrackNb].AX_RACKSTRING[JJ].MesUdcDiffMax_Cell);
				MW(WORD_STRONG:= MesBlock2_Temp[(ParamNbRackString+1)*(KK-1)+JJ+1][ 39], SIGNED:=FALSE, FIX:=3 , SIZE:=1, VAR_OUT := MesDataExd.MesData.AX_RACK[CalrackNb].AX_RACKSTRING[JJ].MesUdc_Cell);
				MW(WORD_STRONG:= MesBlock2_Temp[(ParamNbRackString+1)*(KK-1)+JJ+1][ 40], SIGNED:=FALSE, FIX:=3 , SIZE:=1, VAR_OUT := MesDataExd.MesData.AX_RACK[CalrackNb].AX_RACKSTRING[JJ].MesUdcMax1_Cell);
			MesDataExd.MesData.AX_RACK[CalrackNb].AX_RACKSTRING[JJ].MesUdcMax1_Cell_ModuleID:=MesBlock2_Temp[(ParamNbRackString+1)*(KK-1)+JJ+1][41];
			MesDataExd.MesData.AX_RACK[CalrackNb].AX_RACKSTRING[JJ].MesUdcMax1_Cell_CellID:=MesBlock2_Temp[(ParamNbRackString+1)*(KK-1)+JJ+1][42];
				MW(WORD_STRONG:= MesBlock2_Temp[(ParamNbRackString+1)*(KK-1)+JJ+1][ 43], SIGNED:=FALSE, FIX:=3 , SIZE:=1, VAR_OUT := MesDataExd.MesData.AX_RACK[CalrackNb].AX_RACKSTRING[JJ].MesUdcMin1_Cell);
			MesDataExd.MesData.AX_RACK[CalrackNb].AX_RACKSTRING[JJ].MesUdcMin1_Cell_ModuleID:=MesBlock2_Temp[(ParamNbRackString+1)*(KK-1)+JJ+1][44];
			MesDataExd.MesData.AX_RACK[CalrackNb].AX_RACKSTRING[JJ].MesUdcMin1_Cell_CellID:=MesBlock2_Temp[(ParamNbRackString+1)*(KK-1)+JJ+1][45];
				MW(WORD_STRONG:= MesBlock2_Temp[(ParamNbRackString+1)*(KK-1)+JJ+1][ 46], SIGNED:=FALSE, FIX:=3 , SIZE:=1, VAR_OUT := MesDataExd.MesData.AX_RACK[CalrackNb].AX_RACKSTRING[JJ].MesUdcMax2_Cell);
			MesDataExd.MesData.AX_RACK[CalrackNb].AX_RACKSTRING[JJ].MesUdcMax2_Cell_ModuleID:=MesBlock2_Temp[(ParamNbRackString+1)*(KK-1)+JJ+1][47];
			MesDataExd.MesData.AX_RACK[CalrackNb].AX_RACKSTRING[JJ].MesUdcMax2_Cell_CellID:=MesBlock2_Temp[(ParamNbRackString+1)*(KK-1)+JJ+1][48];
				MW(WORD_STRONG:= MesBlock2_Temp[(ParamNbRackString+1)*(KK-1)+JJ+1][ 49], SIGNED:=FALSE, FIX:=3 , SIZE:=1, VAR_OUT := MesDataExd.MesData.AX_RACK[CalrackNb].AX_RACKSTRING[JJ].MesUdcMin2_Cell);
			MesDataExd.MesData.AX_RACK[CalrackNb].AX_RACKSTRING[JJ].MesUdcMin2_Cell_ModuleID:=MesBlock2_Temp[(ParamNbRackString+1)*(KK-1)+JJ+1][50];
			MesDataExd.MesData.AX_RACK[CalrackNb].AX_RACKSTRING[JJ].MesUdcMin2_Cell_CellID:=MesBlock2_Temp[(ParamNbRackString+1)*(KK-1)+JJ+1][51];
				MW(WORD_STRONG:= MesBlock2_Temp[(ParamNbRackString+1)*(KK-1)+JJ+1][ 52], SIGNED:=FALSE, FIX:=2 , SIZE:=1, VAR_OUT := MesDataExd.MesData.AX_RACK[CalrackNb].AX_RACKSTRING[JJ].MesTempDiffMax_Cell);
				MW(WORD_STRONG:= MesBlock2_Temp[(ParamNbRackString+1)*(KK-1)+JJ+1][ 53], SIGNED:=TRUE, FIX:=2 , SIZE:=1, VAR_OUT := MesDataExd.MesData.AX_RACK[CalrackNb].AX_RACKSTRING[JJ].MesTemp_Cell);
				MW(WORD_STRONG:= MesBlock2_Temp[(ParamNbRackString+1)*(KK-1)+JJ+1][ 54], SIGNED:=TRUE, FIX:=2 , SIZE:=1, VAR_OUT := MesDataExd.MesData.AX_RACK[CalrackNb].AX_RACKSTRING[JJ].MesTempmax1_Cell);
			MesDataExd.MesData.AX_RACK[CalrackNb].AX_RACKSTRING[JJ].MesTempmax1_Cell_ModuleID:=MesBlock2_Temp[(ParamNbRackString+1)*(KK-1)+JJ+1][55];
			MesDataExd.MesData.AX_RACK[CalrackNb].AX_RACKSTRING[JJ].MesTempmax1_Cell_CellID:=MesBlock2_Temp[(ParamNbRackString+1)*(KK-1)+JJ+1][56];
				MW(WORD_STRONG:= MesBlock2_Temp[(ParamNbRackString+1)*(KK-1)+JJ+1][ 57], SIGNED:=TRUE, FIX:=2 , SIZE:=1, VAR_OUT := MesDataExd.MesData.AX_RACK[CalrackNb].AX_RACKSTRING[JJ].MesTempmin1_Cell);
			MesDataExd.MesData.AX_RACK[CalrackNb].AX_RACKSTRING[JJ].MesTempmin1_Cell_ModuleID:=MesBlock2_Temp[(ParamNbRackString+1)*(KK-1)+JJ+1][58];
			MesDataExd.MesData.AX_RACK[CalrackNb].AX_RACKSTRING[JJ].MesTempmin1_Cell_CellID:=MesBlock2_Temp[(ParamNbRackString+1)*(KK-1)+JJ+1][59];
				MW(WORD_STRONG:= MesBlock2_Temp[(ParamNbRackString+1)*(KK-1)+JJ+1][ 60], SIGNED:=TRUE, FIX:=2 , SIZE:=1, VAR_OUT := MesDataExd.MesData.AX_RACK[CalrackNb].AX_RACKSTRING[JJ].MesTempmax2_Cell);
			MesDataExd.MesData.AX_RACK[CalrackNb].AX_RACKSTRING[JJ].MesTempmax2_Cell_ModuleID:=MesBlock2_Temp[(ParamNbRackString+1)*(KK-1)+JJ+1][61];
			MesDataExd.MesData.AX_RACK[CalrackNb].AX_RACKSTRING[JJ].MesTempmax2_Cell_CellID:=MesBlock2_Temp[(ParamNbRackString+1)*(KK-1)+JJ+1][62];
				MW(WORD_STRONG:= MesBlock2_Temp[(ParamNbRackString+1)*(KK-1)+JJ+1][ 63], SIGNED:=TRUE, FIX:=2 , SIZE:=1, VAR_OUT := MesDataExd.MesData.AX_RACK[CalrackNb].AX_RACKSTRING[JJ].MesTempmin2_Cell);
			MesDataExd.MesData.AX_RACK[CalrackNb].AX_RACKSTRING[JJ].MesTempmin2_Cell_ModuleID:=MesBlock2_Temp[(ParamNbRackString+1)*(KK-1)+JJ+1][64];
			MesDataExd.MesData.AX_RACK[CalrackNb].AX_RACKSTRING[JJ].MesTempmin2_Cell_CellID:=MesBlock2_Temp[(ParamNbRackString+1)*(KK-1)+JJ+1][65];
				MW(WORD_STRONG:= MesBlock2_Temp[(ParamNbRackString+1)*(KK-1)+JJ+1][ 66], SIGNED:=TRUE, FIX:=2 , SIZE:=1, VAR_OUT := MesDataExd.MesData.AX_RACK[CalrackNb].AX_RACKSTRING[JJ].MesTempPCBMax);
			MesDataExd.MesData.AX_RACK[CalrackNb].AX_RACKSTRING[JJ].MesTempPCBMax_ModuleID:=MesBlock2_Temp[(ParamNbRackString+1)*(KK-1)+JJ+1][67];
				MW(WORD_STRONG:= MesBlock2_Temp[(ParamNbRackString+1)*(KK-1)+JJ+1][ 68], SIGNED:=TRUE, FIX:=2 , SIZE:=1, VAR_OUT := MesDataExd.MesData.AX_RACK[CalrackNb].AX_RACKSTRING[JJ].MesTempPCBMin);
			MesDataExd.MesData.AX_RACK[CalrackNb].AX_RACKSTRING[JJ].MesTempPCBMin_ModuleID:=MesBlock2_Temp[(ParamNbRackString+1)*(KK-1)+JJ+1][69];
			MesDataExd.MesData.AX_RACK[CalrackNb].AX_RACKSTRING[JJ].MesSensorStatus:=MesBlock2_Temp[(ParamNbRackString+1)*(KK-1)+JJ+1][75];
			MesDataExd.MesData.AX_RACK[CalrackNb].AX_RACKSTRING[JJ].MesModuleScanStatus:=MesBlock2_Temp[(ParamNbRackString+1)*(KK-1)+JJ+1][76];
			MesDataExd.MesData.AX_RACK[CalrackNb].AX_RACKSTRING[JJ].MesModuleBalancingStatus:=MesBlock2_Temp[(ParamNbRackString+1)*(KK-1)+JJ+1][77];
			MesDataExd.MesData.AX_RACK[CalrackNb].AX_RACKSTRING[JJ].MesModuleAddressStatus:=MesBlock2_Temp[(ParamNbRackString+1)*(KK-1)+JJ+1][78];
			MesDataExd.MesData.AX_RACK[CalrackNb].AX_RACKSTRING[JJ].MesModuleVoltageStatus:=MesBlock2_Temp[(ParamNbRackString+1)*(KK-1)+JJ+1][79];
			MesDataExd.MesData.AX_RACK[CalrackNb].AX_RACKSTRING[JJ].MesModuleTemperatureStatus:=MesBlock2_Temp[(ParamNbRackString+1)*(KK-1)+JJ+1][80];
			MesDataExd.MesData.AX_RACK[CalrackNb].AX_RACKSTRING[JJ].MesState:=MesBlock2_Temp[(ParamNbRackString+1)*(KK-1)+JJ+1][87];
				
				MW(WORD_STRONG:= MesBlock2_Temp[(ParamNbRackString+1)*(KK-1)+JJ+1][ 81], 	SIGNED:=FALSE, FIX:=2 , SIZE:=1, VAR_OUT := MesDataExd.MesData.AX_RACK[CalrackNb].AX_RACKSTRING[JJ].MesUdcDiffCellMax);
				MW(WORD_STRONG:= MesBlock2_Temp[(ParamNbRackString+1)*(KK-1)+JJ+1][ 82], 	SIGNED:=FALSE, FIX:=2 , SIZE:=1, VAR_OUT := MesDataExd.MesData.AX_RACK[CalrackNb].AX_RACKSTRING[JJ].MesUdcDiffModuleMax);
			MesDataExd.MesData.AX_RACK[CalrackNb].AX_RACKSTRING[JJ].MesUdcDiffModuleMax_ModuleID:=MesBlock2_Temp[(ParamNbRackString+1)*(KK-1)+JJ+1][83];
				MW(WORD_STRONG:= MesBlock2_Temp[(ParamNbRackString+1)*(KK-1)+JJ+1][ 84], 	SIGNED:=FALSE, FIX:=2 , SIZE:=1, VAR_OUT := MesDataExd.MesData.AX_RACK[CalrackNb].AX_RACKSTRING[JJ].MesUdcDiffCellMin);
				MW(WORD_STRONG:= MesBlock2_Temp[(ParamNbRackString+1)*(KK-1)+JJ+1][ 85], 	SIGNED:=FALSE, FIX:=2 , SIZE:=1, VAR_OUT := MesDataExd.MesData.AX_RACK[CalrackNb].AX_RACKSTRING[JJ].MesUdcDiffModuleMin);
			MesDataExd.MesData.AX_RACK[CalrackNb].AX_RACKSTRING[JJ].MesUdcDiffModuleMin_ModuleID:=MesBlock2_Temp[(ParamNbRackString+1)*(KK-1)+JJ+1][86]	;
				MW(WORD_STRONG:= MesBlock2_Temp[(ParamNbRackString+1)*(KK-1)+JJ+1][ 88], 	SIGNED:=FALSE, FIX:=0 , SIZE:=1, VAR_OUT := MesDataExd.MesData.AX_RACK[CalrackNb].AX_RACKSTRING[JJ].MesCellVDist_under20mV);
				MW(WORD_STRONG:= MesBlock2_Temp[(ParamNbRackString+1)*(KK-1)+JJ+1][ 89], 	SIGNED:=FALSE, FIX:=0 , SIZE:=1, VAR_OUT := MesDataExd.MesData.AX_RACK[CalrackNb].AX_RACKSTRING[JJ].MesCellVDist_underVimbAlarm );
				MW(WORD_STRONG:= MesBlock2_Temp[(ParamNbRackString+1)*(KK-1)+JJ+1][ 90], 	SIGNED:=FALSE, FIX:=0 , SIZE:=1, VAR_OUT := MesDataExd.MesData.AX_RACK[CalrackNb].AX_RACKSTRING[JJ].MesCellVDist_underVimbProtection );
				MW(WORD_STRONG:= MesBlock2_Temp[(ParamNbRackString+1)*(KK-1)+JJ+1][ 91], 	SIGNED:=FALSE, FIX:=0 , SIZE:=1, VAR_OUT := MesDataExd.MesData.AX_RACK[CalrackNb].AX_RACKSTRING[JJ].MesCellVDist_VimbProtection );
			MesDataExd.MesData.AX_RACK[CalrackNb].AX_RACKSTRING[JJ].MesCellBalancingCntMax:=MesBlock2_Temp[(ParamNbRackString+1)*(KK-1)+JJ+1][92];
			MesDataExd.MesData.AX_RACK[CalrackNb].AX_RACKSTRING[JJ].MesCellBalancingCntMax_ModuleID:=MesBlock2_Temp[(ParamNbRackString+1)*(KK-1)+JJ+1][93];
			MesDataExd.MesData.AX_RACK[CalrackNb].AX_RACKSTRING[JJ].MesCellBalancingCntMax_CellID:=MesBlock2_Temp[(ParamNbRackString+1)*(KK-1)+JJ+1][94];
				MW(WORD_STRONG:= MesBlock2_Temp[(ParamNbRackString+1)*(KK-1)+JJ+1][ 95], Word_WEAK:= MesBlock2_Temp[(ParamNbRackString+1)*(KK-1)+JJ+1][96], 	SIGNED:=FALSE, FIX:=0 , SIZE:=2, VAR_OUT := MesDataExd.MesData.AX_RACK[CalrackNb].AX_RACKSTRING[JJ].MesMaxBalancingTime);

			END_IF
		END_IF


	END_FOR 

END_FOR


SUPER^.M_Read();
END_METHOD

METHOD M_Write
VAR_INPUT
END_VAR
VAR
	InputAddr: WORD;
	KK: INT ;
END_VAR


FOR KK := 1 TO 3 DO
	AX_TrigWrite[KK](CLK := ClockWrite);	
END_FOR

// Si écriture de AX_Cmd[1] -> Commande d'ouverture et de fermeture du DC
IF AX_TrigWrite[1].Q THEN
	IF AX_Cmd[1] = 16#0005 THEN
		CmdCloseDc := TRUE;
		CmdOpenDc := FALSE;
		
	END_IF
	IF AX_Cmd[1] = 16#0003 THEN
		CmdCloseDc := FALSE;
		CmdOpenDc := TRUE;
	END_IF	
END_IF

//Si écriture de AX_Cmd[2] -> Commande reset
IF AX_TrigWrite[2].Q THEN
	IF AX_Cmd[2] = 16#0050 THEN
		CmdReset := TRUE;
	END_IF
END_IF
//Si écriture de AX_Cmd[3] -> Watchdog
IF AX_TrigWrite[3].Q THEN
	MesWatchdog := WORD_TO_UINT(AX_Cmd[3]);
END_IF
END_METHOD

END_FUNCTION_BLOCK

// ---- 01_Equipement_Library/Datalogger/FB_Datalogger_Base.TcPOU
FUNCTION_BLOCK FB_Datalogger_Base

VAR_INPUT PERSISTENT
	ParamTcpPort				: UINT	:=	502;		// Modbus TCP port
	ParamIPAddress				: STRING; 				// (NA)Config: IP Adress 
	ParamUnitID					: BYTE;					// (NA)   Modbus Unit ID. 
	ParamID_PTR					: BYTE; 				//ID of the datalogger. Corresponding to PTR ID. 
END_VAR

       	
VAR_INPUT           	
	IN_CmdToggleRead			: BOOL;
	IN_CmdToggleWrite			: BOOL;
	IN_CmdReset_L				: BOOL;
END_VAR             	
      	
VAR                 	
	bInit						: BOOL; 	

//INPUT
	ClockReadInput				: BOOL;							// (NA) Modbus reading Clock
    TP1							: TP ; 							// (NA) Tempo to define Modbus Reading Frequency 
	ParamClockInputTime 		: TIME 		:= TIME#2S;	  		// (Time) Read Modbus Frequency  
	CalCP_Input					: BOOL;
	CalCP_Output				: BOOL;
	
	Trig_Cmd_Read				: R_Trig;
	Trig_Cmd_Write              : R_Trig;
	
	RS_Cmd_Read					: RS;
	RS_Cmd_Write                : RS;
	
	ModbusWriteTimeOut			: TIME;
	FirstTime					: BOOL;

	
//  MesDataExd.MesData.                    : Datalogger;
END_VAR

METHOD M_Execute : BOOL
VAR_INPUT
END_VAR
END_METHOD

END_FUNCTION_BLOCK

// ---- 01_Equipement_Library/Datalogger/FB_Datalogger_PPCVerrerie.TcPOU
FUNCTION_BLOCK FB_Datalogger_PPCVerrerie	EXTENDS FB_Datalogger_Base	// Data from PPC ( MV + HV )
VAR_INPUT PERSISTENT
	// Parameters of the Object (instance specific) 
	ParamTempoComAlarm			: TIME 			:= T#10S ; 						// (s) Config : Tempo to detect LOC Alarm
	ParamClockReadTime 			: TIME 			:= TIME#200MS;	  				// (Time) Read Modbus Frequency.  
	ParamTimeout				: TIME  		:= T#2S ;			  			// (Time) Timeout for modbus reading
	ParamIPAdr : STRING := '192.168.1.2'; // IP Address for Modbus Requests 
END_VAR
VAR_INPUT
	IN_CmdToggleRead			: BOOL ;
	IN_CmdReset_L				: BOOL  ; // Reset Order .
END_VAR
VAR
MesDataExd	AT %Q*				: Datalogger_PPCVerrerie;
	

    Trig_Cmd_Read				: R_TRIG;                       


	
	ClockRead					AT %Q*		: BOOL ;
	
	
	
	
END_VAR

METHOD M_Execute
//////////////////
//  Method Calls 
/////////////////
VAR 
	// Method local variables (reinitialized at each cycle) 
	// EMULATOR

	
END_VAR
END_METHOD

END_FUNCTION_BLOCK

// ---- 01_Equipement_Library/Datalogger/FB_Datalogger_SchSkid.TcPOU
FUNCTION_BLOCK FB_Datalogger_SchSkid EXTENDS FB_Datalogger_Base
 

VAR_INPUT PERSISTENT

	ParamTempoComAlarm			: TIME 		:= T#30S ; 							// (s) Config : Tempo to detect LOC Alarm
	ParamTimeOutCurtail     	: TIME 		:= T#45S ;							// (s) Config : Tempo to curtail power at set value before Timeout warning
	ParamClockReadTime 			: TIME 		:= TIME#11S;	  					// (Time) Read Modbus Frequency . 
	ParamClockWriteTime 		: TIME 		:= TIME#2S; 	  					// (Time) Write Modbus Frequency .
 	ParamTimeout				: TIME  	:= T#5S ;		  					// (Time) Timeout for modbus reading
END_VAR

       	
VAR_INPUT           	
	// I/O Inputs 
	
END_VAR             	
      	
VAR                 	
MesDataExd  AT %Q*		: Datalogger_SchSkid;

    Emul_Pyrano_Value 			: REAL := 10;  
	Emul_TempPanel_Value 		: REAL := 9;	
	Emul_WindSp_Value 			: REAL := 15;
	Emul_WindDir_Value			: REAL := 13;  
            	
	CmdbyCom 		AT %Q*		: WORD;
//INPUT Modbus
	FB_ModbusRead	          	: ARRAY[1..2] OF FB_ModbusRead; 	            // (NA) FB for Modbus Reading
	FB_COMWrite					: FB_ModbusWrite;
	MesBlock1_Temp				: ARRAY [1..19] OF WORD ; 
	MesBlock2_Temp 				: ARRAY [1..26] OF WORD ; 
	
	ModbusInputBoolAlarms		: BOOL;
	ModbusInputBoolAlarmId		: UDINT;
	ModbusInputAnaAlarms		: BOOL;
	ModbusInputAnaAlarmId		: UDINT;
	TEMP_4_20					: ARRAY [1..13] OF REAL;

//OUTPUT Modbus
	MesModbusCmdByComAlarm 		: BOOL;
	MesModbusCmdByComCodeId		: UDINT;
	Front_Montant				: R_Trig;
	RS_Open						: RS;
	RS_Close					: RS;	
END_VAR

METHOD M_Execute : BOOL
VAR_INPUT
END_VAR

// Modeliser les MainMVCB_PTR
//Outputs
IF ParamID_PTR = 1 OR ParamID_PTR = 2 THEN
MesDataExd.MesState_MVCB 				:= 	CmdbyCom.1 OR NOT A1_SUBMV.AX_FeederMVCB[1].IN_MesOpened_IO;
ELSE
MesDataExd.MesState_MVCB 				:= 	CmdbyCom.1 OR NOT A1_SUBMV.AX_FeederMVCB[2].IN_MesOpened_IO;
END_IF


	AX_PTR[ParamID_PTR].A1_MainMVCB_PTR.IN_MesClosed_IO := MesDataExd.MesState_MVCB;




AX_PTR[ParamID_PTR].A1_MainMVCB_PTR.IN_MesComutLocal_IO	:= MesDataExd.MesComutLocal;

// Inputs
//MesDataExd.MesData.MesWatchdog_ProtectRelayVIP  :=	AX_PTR[ParamID_PTR].A1_VIP410.MesDataExd.MesData.MesWatchdog;	// check vip				
MesDataExd.CB_INV[1].MesAlarmState	 	:=	SEL(AX_PTR[ParamID_PTR].MesDataExd.AX_INV[1].MesState = 8 OR AX_PTR[ParamID_PTR].MesDataExd.AX_INV[1].MesState = 5, FALSE, TRUE) OR AX_PTR[ParamID_PTR].MesDataExd.MainMVCB_PTR.MesData.MesOpened;										
MesDataExd.CB_INV[2].MesAlarmState	 	:=	SEL(AX_PTR[ParamID_PTR].MesDataExd.AX_INV[2].MesState = 8 OR AX_PTR[ParamID_PTR].MesDataExd.AX_INV[2].MesState = 5, FALSE, TRUE) OR AX_PTR[ParamID_PTR].MesDataExd.MainMVCB_PTR.MesData.MesOpened;					

IF 	ParamID_PTR	= 4 THEN
MesDataExd.CB_INV[1].MesAlarmState 	:= MesDataExd.CB_INV[2].MesAlarmState; 								// CB of inverter one is in inverter 2
END_IF

MesdataExd.MesComutLocal := TRUE;									
MesDataExd.MesState_MVCB := SEL(AX_PTR[ParamID_PTR].A1_MainMVCB_PTR.IN_MesClosed_IO, FALSE, TRUE); 								
//MesDataExd.MesData.MesFault_ProtectRelayVIP := AX_PTR[ParamID_PTR].A1_VIP410.MesDataExd.MesData.MesAlarmCom;						

//MesDataExd.MesData.Transfo_Synthesis.MesDataExd.MesData.MesAlarmTemp := AX_PTR[ParamID_PTR].A1_Transfo_1.MesDataExd.MesData.MesAlarmTemp OR AX_PTR[ParamID_PTR].A1_Transfo_2.MesDataExd.MesData.MesAlarmTemp;			
//MesDataExd.MesData.Transfo_Synthesis.MesDataExd.MesData.MesAlarmsSynthesis := AX_PTR[ParamID_PTR].A1_Transfo_1.MesDataExd.MesData.MesAlarmsSynthesis OR AX_PTR[ParamID_PTR].A1_Transfo_2.MesDataExd.MesData.MesAlarmsSynthesis;		
MesDataExd.DS_Synthesis.MesAlarmState := FALSE ;							
	
// 4-20 mA
A1_WS.AX_Pyrano[1].IN_MesIOReal1       				:= Emul_Pyrano_Value;    
A1_WS.AX_Pyrano[2].IN_MesIOReal1 					:= Emul_Pyrano_Value;
A1_WS.AX_Pyrano[3].IN_MesIOReal1 					:= Emul_Pyrano_Value;
A1_WS.AX_Pyrano[4].IN_MesIOReal1 					:= Emul_Pyrano_Value;
                                            		
A1_WS.AX_Temp_Panel[1].IN_MesIOReal1  		:= Emul_TempPanel_Value;
A1_WS.AX_Temp_Panel[2].IN_MesIOReal1  		:= Emul_TempPanel_Value;
A1_WS.AX_Temp_Panel[3].IN_MesIOReal1  		:= Emul_TempPanel_Value;
//A1_WS.AX_Temp_Panel[4].IN_MesIOReal1  		:= Emul_TempPanel_Value;
END_METHOD

END_FUNCTION_BLOCK

// ---- 01_Equipement_Library/Datalogger/FB_Datalogger_SENECA.TcPOU
FUNCTION_BLOCK FB_Datalogger_SENECA EXTENDS FB_Datalogger_Base
 

VAR_INPUT PERSISTENT
	ParamWriteTimeout			: TIME  	:= T#5S ;		  					(* (Time) Timeout for modbus reading*)
END_VAR

       	
VAR_INPUT           	
	// I/O Inputs 
	
END_VAR             	
      	
VAR 
MesDataExd				: Datalogger_SENECA;                		
	
//INPUT Modbus
	FB_ModbusRead	          	: ARRAY[1..2] OF FB_ModbusRead; 	            // (NA) FB for Modbus Reading	
	MesBlock1_Temp				: ARRAY [1..8] OF WORD ; 
	
	AlarmModbusInput			: BOOL;
	AlarmID_ModbusInput			: UDINT;
END_VAR

METHOD M_Execute : BOOL
VAR_INPUT
END_VAR

		MesDataExd.MesData.MesWindSp := 14;
		MesDataExd.MesWindDir := 80;
END_METHOD

END_FUNCTION_BLOCK

// ---- 01_Equipement_Library/Fan/FB_Fan_Basic.TcPOU
FUNCTION_BLOCK FB_Fan_Basic
// Function Block to ensure fan control 

VAR_INPUT PERSISTENT
	ParamNbSensors		: INT;					// Number of temperature sensors
	ParamTemphigh 			: REAL := 35;		//  (C)High temperature to trigger the fan
	ParamTemplow 			: REAL := 30;		//  (C)Low temperature to trigger the fan
END_VAR
	
VAR_INPUT           	
	IN_LocalHour     	: TIMESTRUCT;	// 
	IN_ForceRun				: BOOL;		//
	IN_Tmp1_IO 				: REAL;     //  Temperature sensor 1
	IN_Tmp2_IO				: REAL ;    //  Temperature sensor 2

	
	// Commands and setpoints 
	IN_CmdReset_L			: BOOL ;	// (NA) External Reset Command
	
END_VAR             	
VAR_OUTPUT          	
	OUT_Run_IO					: BOOL;
END_VAR             	
VAR                 	
	bInit				: BOOL := TRUE;	// Booleen d'initialisation
	bTmp1_OK			: BOOL; // Booléen de test si les valeurs remontées par les capteurs de températures remontent une donnée correcte
	bTmp2_OK			: BOOL;
	bTmp_OK 			: BOOL;
	fTmp_PT				: REAL;
	// AlarmManagement //

	

	
	// State Mananger //
	MesState			: BYTE;  // Cal 
	
	// M_Evaluate //
	
MesData		: Fan;
END_VAR

VAR PERSISTENT


	MesStartTime 		: WORD := 9;
	MesStopTime 			: WORD := 19;
END_VAR

METHOD M_Execute : BOOL
VAR_INPUT
END_VAR
END_METHOD

END_FUNCTION_BLOCK

// ---- 01_Equipement_Library/GRID/FB_GRID_Base.TcPOU
FUNCTION_BLOCK FB_GRID_Base 
//////////////////
// Grid Operator interface. Base FB.
//////////////////
VAR_INPUT PERSISTENT
	// Parameters of the Object (instance specific) 
	
END_VAR

VAR_INPUT
	// I/O Inputs 
		MesConnectOrderIO			: BOOL ; 					// (NA) 
		MesDisconnectOrderIO 		: BOOL ; 					// (NA) 	
		
END_VAR

VAR_OUTPUT
	//Child objects
	
END_VAR
VAR
	//M_ALARMMANAGEMENT VARIABLES//                                                    								
//	MesDataExd				: GRID ;                   								
		
	//M_INIT VARIABLES //
		bInit						: BOOL:= TRUE ; 			// (NA) Initialize object parameters at first cycle 
		
	// M_EXECUTE VARIABLES //
	
   		MesCP_Read					: BOOL := TRUE;	(* Read function enable *)
END_VAR

METHOD M_CP

VAR 
	// Method local variables (reinitialized at each cycle) 
	
END_VAR
MesCP_GRID := TRUE ;  // Conditions to activate DEIE .
END_METHOD

METHOD M_Evaluate
//////////////////
//  Read Modbus Variable for PCS. 
/////////////////
VAR 
	// Method local variables (reinitialized at each cycle) 
	
END_VAR

///MesDataExd.MesData.:= MesDataExd.MesData.rderInit ; 

IF MesCP_GRID THEN 
MesDataExd.MesData.OUT_CmdAutCpl     := MesConnectOrderIO    ; 
MesDataExd.MesData.OUT_CmdDisconnect := MesDisconnectOrderIO ; 
	
END_IF
END_METHOD

METHOD M_Execute
//////////////////
//  Method Calls 
/////////////////
VAR 
	// Method local variables (reinitialized at each cycle) 

END_VAR

// PERMANENT CONDITIONS //
	M_CP() ; 
	
// METHODS CALLS //
	M_Evaluate() ;
END_METHOD

END_FUNCTION_BLOCK

// ---- 01_Equipement_Library/GRID/FB_GRID_Enedis.TcPOU
FUNCTION_BLOCK FB_GRID_Enedis
//////////////////
// Grid Operator interface . Base FB
//////////////////
VAR_INPUT PERSISTENT
	// Parameters of the Object (instance specific) 
		ParamRseAvailable							: BOOL:=TRUE	; // GRID with RSE option
		ParamTaAvailable							: BOOL:=TRUE	; // GRID with Teleaction option
		ParamP0Available							: BOOL:=TRUE	; // GRID with P regulation option
		ParamQ0Available							: BOOL:=TRUE	; // GRID with Q regulation option
		ParamTONFiltering							: TIME:=T#200MS	; // Minimum tempo filter before command validation (Noise filtering)
		ParamPmaxPark								: REAL;			  //(kW) Contractual maximal power plant active power
		ParamQMax									: REAL;			  // (Kvar)   Contractual maximal power plant reactive power
		ParamQMin									: REAL; 		  // (Kvar)  Contractual maximal power plant reactive power
		ParamPMin									: REAL;			  // (kW) Contractual minimal power plant active power
END_VAR


VAR_INPUT
	// I/O Inputs 
		//FROM ENEDIS
		IN_CmdAutCpl_IO								: BOOL; 	//	Autorisation de couplage
		IN_CmdDisconnect_End_IO						: BOOL; 	//	Fin de demande de decouplage
		IN_CmdDisconnect_IO							: BOOL;		//	Demande de decouplage
		IN_CmdRSEOn_IO								: BOOL;		//	Mise en RSE
		IN_CmdRSEOff_IO								: BOOL;		//	Mise Hors RSE
		IN_CmdTAOn_IO								: BOOL; 	//	Teleaction en service
		IN_CmdTAOff_IO								: BOOL; 	//	Teleaction Hors service
		IN_CmdStopPReg_IO							: BOOL;		//	Fin de passage a P0
		IN_CmdStartPReg_IO							: BOOL;		//	Passage a P0
		IN_CmdStopQReg_IO							: BOOL;		//	Fin de passage a Q0
		IN_CmdStartQreg_IO							: BOOL;		//	Passage a Q0
		IN_CmdEndDisconnectOrder_IO					: BOOL;		//	Fin demande déconnection d'urgence		
		IN_CmdEmergencyDisconnect_IO				: BOOL;		//	Demande d'effacement d'urgence
		IN_CmdEmergencyDisconnect_End_IO			: BOOL; 	//	 Fin demande d'effacement d'urgence	
		IN_CmdDisconnectFromTac_IO					: BOOL; 	//	Decouplage par tac
		IN_CmdTacInFault_IO							: BOOL; 	//	Défaut Tac
		(* 4..20mA *)                                       	
		IN_MesP0Reg_IO								: INT; 		// Kw
		IN_MesQ0Reg_IO								: INT; 		// Kvar
		
		
		//FROM AKSES
		IN_CmdAutCpl_other							: BOOL;
		IN_CmdEmergencyDisconnect_other				: BOOL;
		IN_CmdEmergencyDisconnect_End_other			: BOOL;
		IN_CmdDisconnect_other						: BOOL;
		IN_CmdDisconnect_end_other					: BOOL;
		IN_CmdStartPReg_other						: BOOL;
		IN_CmdStartQReg_other						: BOOL;
		IN_CmdStopPReg_other						: BOOL;
		IN_CmdStopQReg_other						: BOOL;
		
		(*TC Relais Protection*)
		IN_ConnectAuthorizationLost					: BOOL; (*Tous les cas pour un Reset aut Couplage recu*)
		IN_Unavailable								: BOOL; (*Disjoncteur général en Local, ou tous les départs en Local ou Bouton d'arret d'urgence *)
		IN_PP_Connected								: BOOL; (*Centrale Couplée si DG = Fermé et au moins 1 départ antenne en production et au moins un onduleur en Prod*)

END_VAR 


VAR_OUTPUT
		OUT_MesPPUnavailable_IO					: BOOL; // TS centrale indisponible*)
		OUT_MesPPConnected_IO					: BOOL; // Centrale couplée(1)/Centrale Découplée(0)*)
		OUT_MesAutCpl_IO 						: BOOL; // Autorisation de couplage reçue(1)/Attente d'autorisation de couplage(0)*)
		OUT_MesDisconnect_IO 					: BOOL; // Demande de découplage reçue(1)/Fin de demande de découplage(0)*)
		OUT_MesEmergencyDisconnect_IO 			: BOOL; // Demande d effacement d'urgence reçue*)
		OUT_MesRSEON_IO							: BOOL; // Demande mise en RSE reçue*)
		OUT_MesRSEOff_IO						: BOOL; // Demande mise en RSE en attente*)
		OUT_MesTAOn_IO							: BOOL; // Demande mise en TeleAction reçue*)
		OUT_MesTAOff_IO							: BOOL; // Demande mise en TeleAction en attente*)
		OUT_MesStartPReg_IO						: BOOL; // Demande mise en regulation de P reçue*)
		OUT_MesStopPReg_IO						: BOOL; // Demande mise en regulation de P en attente*)
		OUT_MesStartQReg_IO						: BOOL; // Demande mise en regulation de Q reçue*)
		OUT_MesStopQReg_IO						: BOOL; // Demande mise en regulation de Q en attente*)	
	
END_VAR


VAR PERSISTENT
	MesDataExd						: GRID_Enedis;	
END_VAR
VAR
	//M_ALARMMANAGEMENT VARIABLES//                                                    								


	//M_EVALUATE VARIABLES//
		//
		MesDataInit									: GRID_Enedis;					
		//TON                                   	
		TONConnectAuthorization						: TON;
		TONEmergencyDisconnect	               		: TON;
	    TONEmergencyDisconnect_end	            	: TON;
	    TONDisconnect	               				: TON;
	    TONDisconnect_end               	 		: TON;
	    TONPRegOn				                	: TON;
	    TONPRegOff				                	: TON;
	    TONQregOn				                	: TON;
	    TONQRegOff				                	: TON;
	    TONRSEOn				                	: TON;
	    TONRSEOff				                	: TON;
	    TONTAOn					                	: TON;
	    TONTAOff				                	: TON;
		
				
END_VAR

METHOD M_Execute
//////////////////
//  Method Calls 
/////////////////
VAR 
	// Method local variables (reinitialized at each cycle) 
	// EMULATOR

	
END_VAR
END_METHOD

END_FUNCTION_BLOCK

// ---- 01_Equipement_Library/HVAC/FB_HVAC.TcPOU
FUNCTION_BLOCK FB_HVAC
VAR_INPUT PERSISTENT
	ParamIpAddress							: STRING;
	ParamUnitID								: BYTE  	:= 1 ; 
	ParamTcpPort							: UINT 		:= 502;
	ParamPriority							: UINT;
	ParamClockWriteTime						: TIME 		:= T#5S;
	ParamClockReadTime						: TIME 		:= T#5S;
	ParamTimeOut							: TIME 		:= T#2S;
	ParamMaintainPulse						: TIME 		:= T#2S;
END_VAR

VAR_INPUT
	IN_SetptTemp				AT%Q*			: REAL;
	IN_SetptHygro				AT%Q*			: REAL;
	IN_CmdStart								: BOOL;
	IN_CmdStop								: BOOL;
	IN_CmdReset_L							: BOOL;
	IN_CmdToggleRead						: BOOL;
    IN_CmdToggleWrite						: BOOL;
END_VAR

VAR

	//M_CP VARIABLES//
		Trig_Cmd_Read				: R_TRIG;                                                                                        
		Trig_Cmd_Write				: R_TRIG;                                                                                        

		
	//M_READ VARIABLES//
	
		
	MesDataExd			AT%Q*		: HVAC;
		BlockToWrite			AT%Q*		: UINT;		
		ClockWrite				AT%Q*		: BOOL;
		ClockRead				AT%Q*		: BOOL;
	
		
END_VAR
VAR_OUTPUT PERSISTENT
		OUT_State							: BOOL;
        OUT_WorkingHr					: TIME;                  			
END_VAR

METHOD M_Execute : BOOL
VAR_INPUT
END_VAR
END_METHOD

END_FUNCTION_BLOCK

// ---- 01_Equipement_Library/HVAC/FB_HVAC_Base.TcPOU
FUNCTION_BLOCK FB_HVAC_Base
VAR_INPUT PERSISTENT
	ParamClockWriteTime						: TIME 		:= T#2S;	(* Modbus Writing Frequency                 *)
	ParamClockReadTime						: TIME 		:= T#1S;	(* Modbus Reading  Frequency                *)	


END_VAR

VAR_INPUT
		IN_CmdToggleRead						: BOOL;
    IN_CmdToggleWrite						: BOOL;
END_VAR

VAR

	//M_CP VARIABLES//
		Trig_Cmd_Read						: R_TRIG;                                                                                        
		Trig_Cmd_Write						: R_TRIG;                                                                                        

	
		TP1								: TP;
		TP2								: TP;
		TpUpdate						: TP;
		Trig_CmdStart					: R_TRIG;
		Trig_CmdReset					: R_TRIG;
		FTrig_CmdReset					: F_TRIG ; 
		Trig_CmdStop					: R_TRIG;
		WorkingHr						: TIME ; 
	
	///MesDataExd			AT%Q*		: HVAC;
	
		ClockWrite				AT%Q*		: BOOL;
		ClockRead				AT%Q*		: BOOL;
		
		MesCP_Read					: BOOL := TRUE;	(* Read function enable *)
		MesCP_Write					: BOOL := TRUE;	(* Write function enable *)
		
		
		
END_VAR
VAR_OUTPUT PERSISTENT
		OUT_State							: BOOL;
        OUT_WorkingHr						: TIME;                  			
END_VAR

METHOD M_AlarmManagement : BOOL
VAR_INPUT
END_VAR

VAR
	FB_AlarmCodeManager			: FB_AlarmCodeManager ;
END_VAR
END_METHOD

METHOD M_CP : BOOL
VAR_INPUT
END_VAR
Trig_Cmd_Read(CLK:=IN_CmdToggleRead);
Trig_Cmd_Write(CLK:=IN_CmdToggleWrite);
	
IF Trig_Cmd_Read.Q THEN
	IN_CmdToggleRead := FALSE;
	MesCP_Read := NOT MesCP_Read;
END_IF


IF Trig_Cmd_Write.Q THEN
	IN_CmdToggleWrite := FALSE;
	MesCP_Write := NOT MesCP_Write;
END_IF
END_METHOD

METHOD M_Evaluate : BOOL
VAR_INPUT
END_VAR
END_METHOD

METHOD M_Execute : BOOL
VAR_INPUT
END_VAR
TP1(IN:=NOT TP1.Q , PT:= ParamClockWriteTime);
ClockWrite 	:= TP1.Q ;
TP2(IN:=NOT TP2.Q , PT:= ParamClockReadTime);
ClockRead 	:= TP2.Q ;

TpUpdate(IN := NOT TpUpdate.Q, PT := T#5M);
	

	M_Evaluate();
	M_AlarmManagement();
	M_CP();
	M_Write();
	M_Read();
END_METHOD

METHOD M_Read : BOOL
VAR_INPUT
END_VAR
END_METHOD

METHOD M_Write : BOOL
VAR_INPUT
END_VAR
VAR
	WordToWrite		: WORD;
	AX_Addr			: ARRAY[1..3] OF UINT :=[1, 2, 3];
	
END_VAR
END_METHOD

END_FUNCTION_BLOCK

// ---- 01_Equipement_Library/HVAC/FB_HVAC_MADI.TcPOU
FUNCTION_BLOCK FB_HVAC_MADI
VAR_INPUT PERSISTENT
	ParamTempoComAlarm						: TIME 			:= T#10S ; 						// (s) Config : Tempo to detect LOC Alarm
	ParamIpAddress							: STRING;		// IP Address
	ParamUnitID								: BYTE  	:= 1 ; // Modbus Unit ID 
	ParamTcpPort							: UINT 		:= 502;	// Modbus TCP Port
	ParamPriority							: UINT;							// Level of priority in the HVAC pool
	ParamClockWriteTime						: TIME 		:= T#2S;	// Modbus Writing Frequency 
	ParamClockReadTime						: TIME 		:= T#1S;// Modbus Reading  Frequency 
	ParamTimeOut							: TIME 		:= T#3S;	// Modbus Timeout


	
END_VAR

VAR_INPUT	
	IN_SetptTemp				AT %Q*		: REAL:=22;
	IN_SetptHygro							: REAL;
	IN_CmdStart								: BOOL;
	IN_CmdStop								: BOOL;
	IN_CmdReset								: BOOL;

	IN_CmdReleaseStop_OPC					: BOOL ; // Manual Cmd. Non prioritaire sur le mode auto. 
	IN_CmdStop_OPC							: BOOL ; // Manual Cmd .Prioriatire sur le mode auto . Dévérouillage seulement sur ordre de start manual.  
	
	
END_VAR

VAR
	
	MesDataExd					AT %Q*: HVAC_MADI;

	MesDataExd					AT %Q*: HVAC;
		
	
		BlockToWrite				AT %Q*	: BOOL;		
		ClockWrite					AT %Q*	: BOOL;
		ClockRead					AT %Q*	: BOOL;
		
		
END_VAR
VAR_OUTPUT PERSISTENT
	          			
END_VAR

METHOD M_Execute : BOOL
VAR_INPUT
END_VAR
END_METHOD

END_FUNCTION_BLOCK

// ---- 01_Equipement_Library/HVAC/FB_HVAC_Standard.TcPOU
FUNCTION_BLOCK FB_HVAC_Standard EXTENDS FB_HVAC_Base
VAR_INPUT PERSISTENT
	{attribute 'OPC.UA.DA' := '1'} 
	ParamIpAddress							: STRING;
	{attribute 'OPC.UA.DA' := '1'} 
	ParamUnitID								: BYTE  := 1 ; 
	{attribute 'OPC.UA.DA' := '1'}                  
	ParamTcpPort							: UINT 	:= 502;
	ParamPriority							: UINT; 

	ParamTimeOut							: TIME 	:= T#2S;
	ParamMaintainPulse						: TIME 	:= T#2S;
END_VAR

VAR_INPUT
	IN_SetptTemp				AT%Q*		: REAL;
	IN_SetptHygro				AT%Q*		: REAL;
	IN_CmdStart								: BOOL;
	IN_CmdStop								: BOOL;
	IN_CmdReset_L							: BOOL;
	
END_VAR

VAR

                                                                                 
	MesDataExd								: HVAC_Standard ; 
		
	//M_READ VARIABLES//
		WriteSetpt							: FB_ModbusWriteSingleRegister;
		WriteCmd							: FB_ModbusWriteSingleCoil;
		ReadStatus							: FB_ModbusReadCoils;
		

		BlockToWrite			AT%Q*		: UINT;			
		TP_MaintainStart				: TP;
		R_TrigWriteCmd					: R_TRIG;
		F_TrigWriteCmd					: F_TRIG;

		R_TrigState						: R_TRIG;
		F_TrigState						: F_TRIG;
		TimeStart						: TIME;
		TimeNotStart					: TIME;
		
END_VAR

METHOD M_AlarmManagement : BOOL
VAR_INPUT
END_VAR

VAR
	FB_AlarmCodeManager			: FB_AlarmCodeManager ;
END_VAR
	FB_AlarmCodeManager(
		bAlarm1			:= FALSE, 	// CB of the battery charger is opened
		bAlarm2			:= FALSE,			// Main switch of tgbt is opened
		bAlarm3			:= False,	// No Voltage on the 48V TGBT
		bAlarm4			:= False,
		bAlarm5			:= False,
		bAlarm6			:= False,
		bAlarm7			:= False,
		bAlarm8			:= False,
		bAlarm9			:= False,
		bAlarm10		:= False,
		bAlarm11		:= False,
		bAlarm12		:= False,
		bAlarm13		:= False,
		bAlarm14		:= False,
		bAlarm15		:= False,
		wAlarmCode		=>MesDataExd.MesData.MesAlarmCode); 
		

// WARNING CODE //
	FB_AlarmCodeManager
(
 		bAlarm1			:= FALSE,
		bAlarm2			:= False,
		bAlarm3			:= False,
		bAlarm4			:= False,
		bAlarm5			:= False,
		bAlarm6			:= False,
		bAlarm7			:= False,
		bAlarm8			:= False,
		bAlarm9			:= False,
		bAlarm10		:= False,
		bAlarm11		:= False,
		bAlarm12		:= False,
		bAlarm13		:= False,
		bAlarm14		:= False,
		bAlarm15		:= False,
		wAlarmCode		=>MesDataExd.MesData.MesWarningCode					
);
END_METHOD

METHOD M_Evaluate : BOOL
VAR_INPUT
END_VAR
END_METHOD

METHOD M_Read : BOOL
VAR_INPUT
END_VAR
ReadStatus
(
	pDestAddr := ADR(OUT_State),
	sIPAddr := ParamIpAddress,
	tTimeout := ParamTimeOut,
	nTcpPort := ParamTcpPort,
	nQuantity := 1,
	nMBAddr := 2,
	cbLength := SIZEOF(OUT_State),
	ClockRead := ClockRead AND MesCP_Read,
	nUnitID := ParamUnitID
);

R_TrigState(CLK := OUT_State AND TpUpdate.Q);
F_TrigState(CLK := OUT_State AND TpUpdate.Q);

IF R_TrigState.Q THEN
	TimeStart := TIME();
END_IF
IF F_TrigState.Q  THEN
	TimeNotStart := TIME();
	OUT_WorkingHr := OUT_WorkingHr + (TimeNotStart-TimeStart);
END_IF
END_METHOD

METHOD M_Write : BOOL
VAR_INPUT
END_VAR
VAR
	WordToWrite		: WORD;
	AX_Addr			: ARRAY[1..3] OF UINT :=[1, 2, 3];
	
END_VAR

WordToWrite := REAL_TO_WORD(IN_SetptTemp*10.0);

Trig_CmdStart(CLK  := IN_CmdStart);
Trig_CmdStop(CLK  := IN_CmdStop);	
Trig_CmdReset(CLk := IN_CmdReset_L);

TP_MaintainStart(IN := Trig_CmdStart.Q OR Trig_CmdStop.Q OR Trig_CmdReset.Q, PT := ParamMaintainPulse);
R_TrigWriteCmd(CLK := TP_MaintainStart.Q);


IF Trig_CmdStart.Q THEN
	BlockToWrite := 1;
END_IF

IF Trig_CmdStop.Q THEN
	BlockToWrite := 0;
END_IF

IF Trig_CmdReset.Q THEN
	BlockToWrite := 2;
END_IF

WriteSetpt
(
	InputWord := (WordToWrite),
	sIPAddr := ParamIpAddress,
	tTimeout := ParamTimeOut,
	nTCPport := ParamTcpPort,
	nMBAddr := 0,
	cbLength := SIZEOF(WordToWrite),
	nQuantity := 1,
	nUnitID := ParamUnitID,
	WriteCmd := ClockWrite AND MesCP_Write
);


WriteCmd
(
	bValue := TP_MaintainStart.Q,
	sIPAddr := ParamIpAddress,
	tTimeout := ParamTimeOut,
	nTCPport := ParamTcpPort,
	nMBAddr := BlockToWrite,
	nUnitID := ParamUnitID,
	WriteCmd := R_TrigWriteCmd.Q OR F_TrigWriteCmd.Q AND MesCP_Write,
);
END_METHOD

END_FUNCTION_BLOCK

// ---- 01_Equipement_Library/Inverter/FB_INV_1000CP_XT.TcPOU
FUNCTION_BLOCK FB_INV_1000CP_XT EXTENDS FB_INV_Base


VAR_INPUT PERSISTENT
	ParamTcpPort				: UINT	:= 502 ;	// Modbus TCP port
	ParamQn					: REAL;				// (kVAr) Nominal Reactive Power
	ParamIPAddress				: STRING; 			// (NA)Config: IP Adress of PV INverter	
	ParamUnitID 				: BYTE; 			// (NA)   SMA Modbus Unit ID. 
	ParamNumInv					: BYTE;             // Inverter Index  
END_VAR

VAR_INPUT 
	// Parameters of the Object (instance specific) 
	AcknowledgeOrder			: BOOL ;			// Acknowledge fault
	ParamNbInv					: WORD ;			// (NA) Nb of inverters per inverter
	                                                    		
	ParamOptionActivated		: WORD ;			// (NA) Option available on the inverter
	                                                    		
	ParamPRamp					:  REAL:= 0 ;		// (s) duration of the ramp from setpoint to setpoint
	ParamQRamp					:  REAL:= 0 ;		// (s) duration of the ramp from setpoint to setpoint
	ParamPfRamp					:  REAL:= 0 ;		// (s) duration of the ramp from setpoint to setpoint

	IN_MesAcCbOpen_IO				:  BOOL ; 			//Retour cablé Physique des contacteur AC des onduleurs	
	Cmd_SwitchOff				:  BOOL ;		    // etat de DO cablé sur les onduleurs pour les eteindres
END_VAR



VAR
	//M_Acknowledge
		
	// M_ALARMMNGMT VARIABLES //
	
	
	// M_READ VARIABLES//
	MesDataExd		AT %Q*	: INV_1000CP_XT;
		//MesDataExd.MesData.C_Read				:  INV_CC;	
		//MesDataExd.MesData.C_Cmd				:  INV_CC;
		
	
		FB_ModbusRead	          	: ARRAY[1..8] OF FB_ModbusRead; 	            // (NA) FB for Modbus Reading
		FB_ModbusWrite				: ARRAY[1..3] OF FB_ModbusWrite;
		AX_ModbusReadAlarm			: ARRAY[1..9] OF BOOL;
		AX_ModbusReadAlarmId		: ARRAY[1..9] OF UDINT;		
		AX_ModbusWriteAlarm			: ARRAY[1..3] OF BOOL;
		AX_ModbusWriteAlarmId		: ARRAY[1..3] OF UDINT;
		
		
		BlockInit					: WORD;							// First Block : Number of inverters in the PCS
		MesBlock1_Temp 				: ARRAY [1..70] OF WORD ; 		// (NA) Temporary Block with multiple modbus reading (Caution : Double Word variables)
		MesBlock2_Temp 				: ARRAY [1..90] OF WORD ; 		// (NA) Temporary Block with multiple modbus reading (Caution : Double Word variables)
		MesBlock3_Temp 				: ARRAY [1..74] OF WORD ; 		// (NA) Temporary Block with multiple modbus reading (Caution : Double Word variables)
		MesBlock4_Temp 				: ARRAY [1..38] OF WORD ; 		// (NA) Temporary Block with multiple modbus reading (Caution : Double Word variables)
		MesBlock5_Temp 				: ARRAY [1..28] OF WORD ; 		// (NA) Temporary Block with multiple modbus reading (Caution : Double Word variables)
		MesBlock6_Temp				: ARRAY [1..13] OF WORD ;		// (NA) Temporary block with both start commands for each inverter
		MesBlock7_Temp				: ARRAY [1..16] OF WORD ;	
		MesBlock8_Temp				: ARRAY [1..4] OF WORD ;
		
		MesBlockWrite1_Temp 		: WORD ;				    	// (NA) Temporary Block with multiple modbus writing (Caution : Double Word variables)
		MesBlockWrite2_Temp			: WORD ;						// (NA) Temporary Block with multiple modbus writing (Caution : Double Word variables)
		MesBlockWrite3_Temp			: ARRAY [1..2] OF WORD ;
	// M_CURTAIL VARIABLES //
	
		LastCurtailMode				: BOOL:=TRUE ;				// Init at true, to force the first write on inverter
		MesCP_WriteCurtailMode		: BOOL ;
		CurtailModeValue_P			: DWORD ; 					// 1077 := WctlMan : Inverter set setpoint, 1079 := WCtlCom Inverter take the setpoint set by com (plc),303 := OFF
		CurtailModeValue_Q			: DWORD ;					// 303:=OFF,1075:= PFCtlCom,1074:= PFCtlMan,1072 VarCtlCom
		
		MesModbusWriteCode          : UDINT ; 					// (NA) Modbus Write Alarm Code 	
		MesModbusCurtailAlarm		: BOOL ;				   	// (NA) Modbus Write Curtail Alarm 
		
		InvQModeValue				: UINT ;					// Mode of Q power control : 1: Q mod, 2: PF mode, 3: Q(P)
		InvSetptQ					: REAL ;					// (kVAr) setpoint for the reactive power for each inverter
		
	
		InvSetptP					: REAL ;					// (kW) Setpoint for the active power for each inverter
		TEMP						: BOOL ;
	// M_INIT //
		Code_Ctrl_Com 				: UINT := 1079 ;
		
		MesModbusCurtailInitAlarm 	: BOOL ;
		
	// M_STARTSTOP//
		StartStop_RTrig				: R_Trig ;
		StartStop_RTrigIO			: R_Trig ;
		
	// M_CP
		CalCP_Acknowledge			: BOOL ;
		//CalCP_CMD_SetPt				: BOOL; 	  // Write command start;
		CalCP_CMD_StartStop			: BOOL ; 		  // Write command start;
		CalCP_CMD_StartStopIO		: BOOL ; 		  // Write command start;
	// M_STATEMANAGER//
	
	//M_EXECUTE VARIABLES //
		TP_READ						: LTP ;			  //Tempo de cadencement FB Modbus
		RTrig						: R_Trig ; 		  //Front montant sur TP_READ.Q
		ReadBusy					: BOOL ;		 //FB Modbus en busy
		bInit						: BOOL ;
	//EMULATOR VARIABLES //
		
END_VAR

METHOD M_Execute
//////////////////
//  Method Calls 
/////////////////

VAR 
	// Method local variables (reinitialized at each cycle) 

END_VAR


SUPER^.M_Execute() ;
END_METHOD

END_FUNCTION_BLOCK

// ---- 01_Equipement_Library/Inverter/FB_INV_Base.TcPOU
FUNCTION_BLOCK FB_INV_Base
//////////////////

// PV INverter. Base FB. 
//////////////////
VAR_INPUT PERSISTENT
	// Parameters of the Object (instance/model specific) 
	ParamTempoComAlarm					: TIME 		:= T#30S ; 			// (s) Config : Tempo to detect LOC Alarm
	ParamTimeOutCurtail     			: TIME 		:= T#45S ;			// (s) 	Config : Tempo to curtail power at set value before Timeout warning
	ParamClockReadTime 					: TIME 		:= TIME#2S;	  		// (Time) Read Modbus Frequency  
	ParamClockWriteTime 				: TIME 		:= TIME#2S; 	  	// (Time) Write Modbus Frequency
 	ParamTimeout						: TIME  	:= T#5S ;		  	// (Time) Timeout for modbus reading
	                        			
	ParamPn								: REAL;      					// (kW)    Nominal Capacity of SMA SC2750
		
END_VAR

VAR_INPUT
		IN_SetptPlimit					: REAL := 10000;		// (kW) [P,H] Dynamic active Power limit setpoint (curtailing)  
		IN_SetptPlimit_Local			: REAL;					// (kW) [P,H] Dynamic active Power limit setpoint (curtailing)  
		IN_SetptQlimit					: REAL := 2000; 		// Dynamic reactive power setpoints 	
		IN_CmdStart						: BOOL;					// (NA) [P,H] External Start Command
		IN_CmdStop 						: BOOL; 				// (NA) [P,H] External Stop CommAND  
		IN_CmdStop_Local				: BOOL; 				// (NA) [P,H] External Stop Command, only for this inverter
		IN_CmdStart_Local				: BOOL:=TRUE;			// (NA) [P,H] External Start Command, only for this inverter	

		
		IN_CmdToggleRead				: BOOL ;
		IN_CmdToggleWrite				: BOOL ; 
		IN_CmdReset_L					: BOOL ;				// (NA) External Reset Command
END_VAR

VAR
	// M_ALARMMNGMT VARIABLES //
		TON_ComAlarm					: TON ; 				// Tempo before deteting loss of communication. 
	    TON_ComWarning					: TON ; 				// Tempo before detecting loss of communication.                                                	
                                    	 		    	
		MesWarningCom					: BOOL ; 				// (NA) [P,H]  True if bad communication
                                    	
		CalModbusWriteAlarm         	: BOOL ; 				// (NA) Modbus Write Alarm synthesis
                                    	
                                    	
	// M_READ VARIABLES//           	
//	MesDataExd		      	: INV ; 				// (NA) [P,H,B] INV  Data Structure 
                                    	

	// M_CURTAIL VARIABLES //
		FB_CheckCommand1		  		: FB_CheckCommand ; 	// (NA) Functionnal Block to check if Curtail limit Writing Successful
		FB_CheckSetPt		  			: FB_CheckSetPt ; 		// (NA) Functionnal Block to check if Q setpoint Writing Successful
                                    	
		R_TRIG_Curtail					: R_TRIG ;
                                    	
		CalCompareWarningCurtail		: BOOL ; 				// (NA) Curtail failed alarm						
		CalCompareWarningQSetpt			: BOOL ; 				// (NA) Curtail failed alarm						
                                    	
		WriteCmdP 			 			: BOOL;					// Modbus Write Rising Edge 
		WriteCmdQ 			 			: BOOL;					// Modbus Write Rising Edge 
	                                	
                                    	
	// M_STARTSTOP//            		
		Trig_Cmd_Read					: R_TRIG; 
		Trig_Cmd_Write					: R_TRIG;                                    	
		                            	
		RS_Cmd_Read						: RS ; 	
		RS_Cmd_Write					: RS ; 	       	
		Trig_Local_Start				: R_Trig;
		Trig_Local_Stop					: R_Trig;
		Trig_Start						: R_Trig;
		Trig_Stop						: R_Trig;	         
		RS_StartStop					: RS ; 					// (NA) Bistable Function for Start and Stop 
		RS_StartStop_Local				: RS;					// (NA) Bistable Function for Start and Stop local                        	
		                            	
	// M_STATEMANAGER//             	
		MesState						: BYTE; 				// (NA) Cal [P,H,B] Bit 0: OFF , Bit 2 : Feeding Slave 	
                                  
	//M_EXECUTE VARIABLES //
		TP1								: TP ; 					// (NA) Tempo to define Modbus Reading Frequency 
		TP2 							: TP ; 					// (NA) Tempo to define Modbus Writing Frequency
		                                                    	
		ClockRead		AT %Q*			: BOOL;					// (NA) Modbus reading Clock
		ClockWrite 		AT %Q*			: BOOL;					// (NA) Modbus writing Clock 		
		
END_VAR

METHOD M_Execute
//////////////////
//  Method Calls 
/////////////////

VAR 
	// Method local variables (reinitialized at each cycle) 

END_VAR
END_METHOD

END_FUNCTION_BLOCK

// ---- 01_Equipement_Library/Inverter/FB_INV_Sch4400.TcPOU
FUNCTION_BLOCK FB_INV_Sch4400 EXTENDS FB_INV_Base


VAR_INPUT PERSISTENT
	ParamTcpPort						: UINT		:= 502;			//	(NA) TCP port
	ParamQn								: REAL;						// (kVar) Q nominal
	ParamIPAddress						: STRING; 					// (NA)Config: IP Adress of PV INverter	
	ParamUnitID 						: BYTE; 					// (NA)   SMA Modbus Unit ID. 
	ParamNumInv							: BYTE;             		// (NA) number of inverters
	                        			
	ParamPTRNum							: BYTE;             		// (NA)Associated PTR
END_VAR


VAR_INPUT 
	IN_Emul_VacPresent					: BOOL; 		// State = True => presence of voltage, state = False => absence of voltage (to be modified from PTR state)
	IN_Emul_VdcPresent					: BOOL; 		// State = True => presence of voltage, state = False => absence of voltage (to be modified from PTR state)
END_VAR
VAR	
	// M_ALARMMNGMT VARIABLES //
	// M_READ VARIABLES//
	MesDataExd	AT %Q*		: INV_Sch4400;
	MesDataExd_IN					: INV_Sch4400;
	
		bInit							: BOOL := TRUE;
	// M_STATEMANAGER//
	
	//M_EXECUTE VARIABLES //
		Emul_SR							: SR; 
		Emul_ComError					: BOOL ; 
		Emul_MesModbusReadAlarm			: ARRAY[1..2] OF BOOL;
		Emul_AlarmINV					: BOOL ; 
		Emul_Test_AC 					: BOOL;	
		Emul_INV_Offline 				: BOOL;
		Emul_INV_Disable				: BOOL;
		Emul_Online_Var					: BOOL;
		Emul_FaultGnd					: BOOL;
		Emul_StateCBac					: BOOL; // true = CBac is closed, false = CBac is opened 
		Emul_StateCBdc					: BOOL; // true = CBdc is closed, false = CBdc is opened  
		Emul_Event_ID   				: INT;		
							
END_VAR

METHOD M_Execute
//////////////////
//  Method Calls 
/////////////////

VAR 
	// Method local variables (reinitialized at each cycle) 
	SppNum			: UINT;

	SetTempSlope	: REAL;
	KK 				: INT;
	MesEActProd		: INT;
END_VAR

// Emulated variables 
MesDataExd.MesFaultGnd			:= Emul_FaultGnd; 

IN_CmdStop_Local 				:= MesDataExd_IN.MesData.OUT_CmdStop;
IN_CmdStart_Local 				:= MesDataExd_IN.MesData.OUT_CmdStart;

Emul_SR(SET1:= IN_CmdStop OR IN_CmdStop_Local, RESET:=IN_CmdStart OR IN_CmdStart_Local); 

// SppNum:= SEL(ParamUnitID>11 ,1 , 2) ; 

// Inverter's State
IF Emul_INV_Offline THEN 
MesDataExd.MesState		:= 8 ; // Inverter is offline : lost of production
ELSIF Emul_SR.Q1 OR NOT MesDataExd.MesStateCBac THEN   
MesDataExd.MesState		:= 5 ; // Inverter is disabled 	
ELSIF Emul_INV_Disable  THEN
MesDataExd.MesState				:= 5 ; // Inverter is disabled 
ELSIF MesP_INVmppt=0 THEN 
MesDataExd.MesState		:= 8;  // Inverter is offline : lost of production( Night time)
ELSIF Emul_Test_AC THEN
MesDataExd.MesState		:= 7 ; // AC test mode
ELSIF Emul_Online_Var THEN
MesDataExd.MesState		:= 20 ; // Lost of production Online var 
ELSE
MesDataExd.MesState		:= 23; // Online PV. Inverter is online in PV.
END_IF	

// Varibles' values
///MesDataExd.MesData.ParamPn				:= 1200  ; 
MesDataExd.MesData.MesUdc					:= 200 ;
MesDataExd.MesData.MesInsuResistor 			:= 150 ;
MesDataExd.MesEDay							:= 1000; 
MesDataExd.MesData.MesCosPhi				:= 0.95; 
MesDataExd.MesData.MesTemp					:= 32;  
MesDataExd.MesTempExt						:= 25;
MesDataExd.MesSetptCosPhi_CC 				:= 0.98;

MesDataExd.MesSetptP_CC 			:=MesDataExd_IN.MesData.OUT_SetptP; //AX_PTR[ParamPTRNum].IN_SetptPlimit/AX_PTR[ParamPTRNum].ParamNbINV ;		
MesDataExd.MesSetptQ_CC 			:= MesDataExd_IN.MesData.OUT_SetptQ; //AX_PTR[ParamPTRNum].IN_SetptQlimit/AX_PTR[ParamPTRNum].ParamNbINV ;	 	


///MesDataExd.MesData.ParamTP_RampP 		:= ;    	
///MesDataExd.MesData.ParamTP_RampQ 		:= ;    	
///MesDataExd.MesData.ParamTP_RampCosPhi 	:= ;  
MesDataExd.MesStartDisabledPersis   := TRUE; 	// By default enable inverter after a power on

// Evaluated variables	
//MesDataExd.MesData.ParamPn 		:= ParamPn; 
MesDataExd.MesData.MesAlarmCom					:= TON_ComAlarm.Q; 					 // find the modbus variable that coresponds to this 
MesDataExd.MesStateCom  			:= NOT MesDataExd.MesData.MesAlarmCom; 
	
SetTempSlope 						:= SEL(MesDataExd.MesData.MesAlarmCom, MesDataExd.MesSetptP_CC, MesDataExd_IN.MesData.ParamPn); 

MesDataExd.MesData.MesP 			:= SEL((A1_PP.MesState =9) OR Emul_AlarmINV OR NOT(AX_PTR[ParamPTRNum].A1_Datalogger.MesDataExd.MesState_MVCB) OR MesDataExd.MesState=5 OR MesDataExd.MesState=8, MIN(SetTempSlope, MesP_INVmppt), 0); 
IN_SetptQlimit						:= MesDataExd_IN.MesData.OUT_SetptQ; 
MesDataExd.MesData.MesQ 			:= IN_SetptQlimit; 
MesDataExd.MesData.MesPdc 			:= MesDataExd.MesData.MesP/0.95; 
MesDataExd.MesData.MesIdc 			:= MesDataExd.MesData.MesPdc/MesDataExd.MesData.MesUdc; 

MesDataExd.MesData.MesU 			:= SEL(MesDataExd.MesState =5 OR MesDataExd.MesState =8 OR NOT IN_Emul_VacPresent, 400, 0); 
MesDataExd.MesData.MesV			    := MesDataExd.MesData.MesU/SQRT(3)*2 ; 
MesDataExd.MesData.MesI			    := SEL(MesDataExd.MesData.MesU = 0 , MesDataExd.MesData.MesP*1000 / MesDataExd.MesData.MesU /SQRT(3) ,0 ) ; 
MesDataExd.MesData.MesFreq			:= A1_SUBMV.A1_PM.MesDataExd.MesData.Mesfreq; 
MesDataExd.MesData.MesS			    := SQRT(MesDataExd.MesData.MesP*MesDataExd.MesData.MesP+MesDataExd.MesData.MesQ*MesDataExd.MesData.MesQ) ; 

// Properties update 
//MesDataExd.MesData.MesAlarmCom		:= MesDataExd.MesData.MesIDState =  ;

MesDataExd.MesI1					:= MesDataExd.MesData.MesI; 
MesDataExd.MesI2					:= MesDataExd.MesData.MesI; 
MesDataExd.MesI3					:= MesDataExd.MesData.MesI; 
MesDataExd.MesU12					:= MesDataExd.MesData.MesU ; 
MesDataExd.MesU23					:= MesDataExd.MesData.MesU ; 
MesDataExd.MesU31					:= MesDataExd.MesData.MesU ; 
MesDataExd.MesV1					:= MesDataExd.MesData.MesV; 
MesDataExd.MesV2					:= MesDataExd.MesData.MesV;  
MesDataExd.MesV3					:= MesDataExd.MesData.MesV; 

MesDataExd.MesData.MesI 			:= (MesDataExd.MesI1 + MesDataExd.MesI2 + MesDataExd.MesI3)/3;
MesDataExd.MesData.MesV 			:= (MesDataExd.MesV1 + MesDataExd.MesV2 + MesDataExd.MesV3)/3;
MesDataExd.MesData.MesS 			:= SQRT(MesDataExd.MesData.MesP*MesDataExd.MesData.MesP + MesDataExd.MesData.MesQ*MesDataExd.MesData.MesQ);


// Energy
IF MesDataExd.MesData.MesP > 0 THEN
MesDataExd.MesEActProd := MesDataExd.MesEActProd + MesDataExd.MesData.MesP*ParamCycleTime_Emul/3600000;
END_IF
IF MesDataExd.MesData.MesP < 0 THEN
MesDataExd.MesEActCons := MesDataExd.MesEActCons - MesDataExd.MesData.MesP*ParamCycleTime_Emul/3600000;
END_IF
IF MesDataExd.MesData.MesQ > 0 THEN
MesDataExd.MesEReactProd := MesDataExd.MesEReactProd + MesDataExd.MesData.MesQ*ParamCycleTime_Emul/3600000;
END_IF
IF MesDataExd.MesData.MesQ < 0 THEN
MesDataExd.MesEReactCons := MesDataExd.MesEReactCons - MesDataExd.MesData.MesQ*ParamCycleTime_Emul/3600000;
END_IF
	                                
MesDataExd.MesStateCBac			:= Emul_StateCBac OR IN_Emul_VacPresent;
MesDataExd.MesStateCBdc			:= Emul_StateCBdc OR IN_Emul_VdcPresent;
	///MesDataExd.MesData.MesStateNoAlert	:=  SEL(Emul_FaultGnd OR ..,1,0); // 1: no alert                                     
	///MesDataExd.MesData.MesBdrigeCtlMod	:= 

// Strings 



MesDataExd.STR[5].MesIdc	:= MesDataExd.MesData.MesIdc/9;  	
MesDataExd.STR[6].MesIdc	:= MesDataExd.MesData.MesIdc/9;	
MesDataExd.STR[7].MesIdc	:= MesDataExd.MesData.MesIdc/9;	
MesDataExd.STR[8].MesIdc 	:= MesDataExd.MesData.MesIdc/9;	
MesDataExd.STR[9].MesIdc	:= MesDataExd.MesData.MesIdc/9;	
MesDataExd.STR[10].MesIdc	:= MesDataExd.MesData.MesIdc/9;	 

		

	
MesDataExd.MesStartDisabled := SEL(MesDataExd.MesState=5 OR MesDataExd.MesState=8 , TRUE, FALSE);

	///MesDataExd.MesData.MesEvendID	    	:= Emul_Event_ID;		  
	///MesDataExd.MesData.MesEventID_Stop		:= ;	  
	///MesDataExd.MesData.MesStateID_Recovery   := ;	  
MesDataExd.MesEventID_AbnormalOff 	:= SEL(MesDataExd.MesState=8 OR MesDataExd.MesState=5,0,Emul_Event_ID);
END_METHOD

END_FUNCTION_BLOCK

// ---- 01_Equipement_Library/Inverter/FB_INV_Smartlogger.TcPOU
FUNCTION_BLOCK FB_INV_Smartlogger EXTENDS FB_INV_Base
//////////////////
// SmartLogger Huawei
//////////////////

VAR 
		KK_ModbusRead					: BYTE;	
		Emul_Smooth						: ARRAY[1..CstNbInv_PTR_G] OF FB_Smooth ; 
		Emul_MesModbusReadAlarm			: ARRAY[1..CstNbInv_PTR_G] OF BOOL;
		Emul_MesModbusReadAlarm2		: BOOL ; 
		Emul_MesModbusReadAlarm3		: BOOL ; 
		Emul_AlarmINV					: BOOL ; 
		Emul_ComError					: BOOL ; 
	
		Emul_MesModbusCurtailAlarm		: BOOL;	
		Emul_RS							: SR; 
END_VAR


VAR_INPUT PERSISTENT
	// Parameters of the Object (instance specific) 
	ParamIPAdress		   : STRING 	:= '127.0.0.1'; 	// (NA)Config: IP Adress of PV INverter

	ParamUnitID 			: BYTE  := 0; 			  // (NA)   Modbus Unit ID. 
	ParamNbINV				: BYTE:=1 ; // Number of inverters behind the smartlogger 
	ParamnTcpPort			: UINT := 502;	// TCP port number 
	ParamPnomINV			: REAL:=60; // (kW) Nominal Power For one inverter 
	ParamSLNum				: BYTE ; 			// (NA) Config :Numerous of the ESS in the PP
			
END_VAR

VAR_OUTPUT
	//Child objects
	
END_VAR

VAR
	// M_ALARMMNGMT VARIABLES //
	                                     		
	
	// M_READ VARIABLES//

	MesDataExd	AT %Q*		: SL_Huawei;

//		FB_ModbusRead_I1          	: ARRAY[1..CstNbINVperPTR_G] OF  FB_ModbusRead ; 	// (NA) FB for Modbus Reading
		FB_ModbusRead_I2          	: FB_ModbusRead ; 	// (NA) FB for Modbus Reading
		FB_ModbusRead_I3          	: FB_ModbusRead ; 	// (NA) FB for Modbus Reading
			
//		MesBlock1_Temp 				: ARRAY[1..CstNbINVperPTR_G] OF ARRAY[0..24]  OF WORD; 			// (NA) Temporary Block with multiple modbus reading (Caution : Double Word variables)
//		MesBlock1_Temp 				: ARRAY[0..25*CstNbINVperPTR_G-1]  OF WORD; 			// (NA) Temporary Block with multiple modbus reading (Caution : Double Word variables)
		MesBlock2_Temp 				: ARRAY[0..56] OF WORD;				// (NA) Temporary Block with multiple modbus reading (Caution : Double Word variables)
		MesBlock3_Temp 				: ARRAY[0..14] OF WORD;				// (NA) Temporary Block with multiple modbus reading (Caution : Double Word variables)

		
//		MesModbusReadAlarm 		  	: ARRAY[1..CstNbINVperPTR_G] OF BOOL ; 			// (NA) Modbus Read Alarm for all modbus frames		
		MesModbusReadAlarm2 		: BOOL ; 			// (NA) Modbus Read Alarm for all modbus frames			
		MesModbusReadAlarm3 		: BOOL ; 			// (NA) Modbus Read Alarm for all modbus frames			

//		MesModbusAlarmCode			: ARRAY[1..CstNbINVperPTR_G] OF UDINT;							// (NA) Modbus Read Alarm Code
		MesModbusAlarmCode2			: UDINT;							// (NA) Modbus Read Alarm Code
		MesModbusAlarmCode3			: UDINT;							// (NA) Modbus Read Alarm Code

	
	// M_CURTAIL VARIABLES //
		FB_ModbusWrite_I2 		  	: FB_ModbusWrite ; 			// (NA) Functionnal Block for Writing Curtail limit through modbus	
		MesModbusWriteCode          : UDINT ; 							// (NA) Modbus Write Alarm Code 	
		
		MesModbusCurtailAlarm		: BOOL ;				   			// (NA) Modbus Write Curtail Alarm 
		WriteBlock_Temp 	AT %Q*					: ARRAY[0..3] OF WORD; 	// Temporary Block with multiple modbus writing	 
			
	// M_STARTSTOP//

	// M_STATEMANAGER//
	
	//M_EXECUTE VARIABLES //



END_VAR

METHOD M_Execute
//////////////////
//  Method Calls 
/////////////////

VAR 
	// Method local variables (reinitialized at each cycle) 

END_VAR

MesDataExd.MesEff			            := 0.9 ; 
MesDataExd.MesData.MesTemp				:= 25 ; 


	MesDataExd.MesData.MesP 			:= 0; 			

		FOR KK_ModbusRead:=1 TO ParamNbINV DO

			Emul_RS(SET1:= IN_CmdStop, RESET:=IN_CmdStart ) ; 
			IF Emul_AlarmINV  THEN 
			MesDataExd.MesData.MesIDState		:= 6 ; 
			ELSIF Emul_RS.Q1 THEN 
			MesDataExd.MesData.MesIDState		:= 0 ;
			ELSIF MesP_INVmppt=0 THEN 

			MesDataExd.MesData.MesIDState		:= 5 ;
			ELSIF IN_SetptPlimit < ParamPnomINV THEN 
			MesDataExd.MesData.MesIDState		:= 3 ; 
			MesDataExd.MesData.MesOn		:= TRUE; 
			ELSIF Emul_ComError THEN 
			MesDataExd.MesData.MesIDState		:= 7 ; 
			ELSE
			MesDataExd.MesData.MesIDState		:= 1 ; 
			MesDataExd.MesData.MesOn			:= TRUE; 
			END_IF	
			


			// Aggregate 
		MesDataExd.MesData.MesP 			:= MesDataExd.MesData.MesP +AX_PTR[ParamSLNum].AX_INV[KK_ModbusRead].MesDataExd.MesData.MesP ; 
			
		END_FOR
		
			
		
	MesDataExd.MesData.MesPdc			:= MesDataExd.MesData.MesP //MesDataExd.MesData.MesEff; 
	MesDataExd.MesData.MesQ		    :=  IN_SetptQlimit; 
	MesDataExd.MesData.MesIdc 		:= MesDataExd.MesData.MesPdc/AX_PTR[ParamSLNum].AX_INV[1].MesDataExd.MesData.MesUdc;  

	MesDataExd.MesData.MesCosPhi			:=SEL( MesDataExd.MesData.MesP > 0.01 , 1 ,  COS.MesDataExd.MesData.MesQ MesDataExd.MesData.MesP ) ) ; 
	

	MesDataExd.MesData.MesU12			:=  A1_SUBMV.A1_PM.MesDataExd.MesData.MesU12 ; 
	MesDataExd.MesData.MesU23			:=  A1_SUBMV.A1_PM.MesDataExd.MesData.MesU23 ;  
	MesDataExd.MesData.MesU31			:=  A1_SUBMV.A1_PM.MesDataExd.MesData.MesU31 ; 
	MesDataExd.MesData.MesI1			:= SEL.MesDataExd.MesData.MesU12= 0 , MesDataExd.MesData.MesP*1000 MesDataExd.MesData.MesU12/SQRT(3) ,0 ) ; 
	MesDataExd.MesData.MesI2			:= MesDataExd.MesData.MesI1  ; 
	MesDataExd.MesData.MesI3			:= MesDataExd.MesData.MesI1 ; 
		
		
	MesDataExd.MesData.MesSetptPMax 	:= ParamPn ; 
	MesDataExd.MesData.MesSetptQMax 	:= 0.6*ParamPn ; 
	MesDataExd.MesData.MesSetptQMin	:= -0.6*ParamPn  ; 
		


MesDataExd.MesData.MesEDay			            := MesDataExd.MesData.MesEDay + MesDataExd.MesData.MesP*ParamCycleTime_Emul/3600000	;
	IF CalLocalTimeStruct.wHour = 1 AND CalLocalTimeStruct.wMinute = 0 AND ParamCycleTime_Emul = 10 THEN
	MesDataExd.MesData.MesEDay	:=0 ;
	END_IF
	
MesDataExd.MesData.MesETot			            := MesDataExd.MesData.MesETot + MesDataExd.MesData.MesP*ParamCycleTime_Emul/3600000	;
END_METHOD

END_FUNCTION_BLOCK

// ---- 01_Equipement_Library/Inverter/FB_INV_Sun2000KtlMo.TcPOU
FUNCTION_BLOCK FB_INV_Sun2000KtlMo EXTENDS FB_INV_Base
VAR 
		KK_ModbusRead					: BYTE;	
		
		Emul_MesModbusReadAlarm			: ARRAY[1..2] OF BOOL;
		Emul_AlarmINV					: BOOL ; 
		Emul_Smooth						: FB_Smooth ;
END_VAR
VAR_INPUT PERSISTENT
	// Parameters of the Object (instance specific) 
	ParamIPAdress	   : STRING := '127.0.0.1'; 	// (NA)Config: IP Adress of PV INverter
	ParamnTcpPort		: UINT := 502;	
	ParamUnitID 		: BYTE  := 1; 	  			// (NA)   SMA Modbus Unit ID. 
	ParamID_INV			: BYTE ; 		        	// (NA) Config :Numerous of the ESS in the PP

END_VAR

VAR_OUTPUT
	//Child objects

END_VAR

VAR
	//M_Acknowledge
		
	// M_ALARMMNGMT VARIABLES //
	MesAlarmCode1			: WORD ; 
	MesAlarmCode2			: WORD ; 
	
	// M_READ VARIABLES//
		Trig_Read					: R_TRIG;

		FB_ModbusRead_I2          	: FB_ModbusRead ; 	// (NA) FB for Modbus Reading
		FB_ModbusRead_I3          	: FB_ModbusRead ; 	// (NA) FB for Modbus Reading

		MesBlock_Temp 				: ARRAY[1..2] OF ARRAY [1..125] OF WORD ; 			// (NA) Temporary Block with multiple modbus reading (Caution : Double Word variables)

		AX_Busy						: ARRAY[1..2] OF BOOL;
		AX_Error					: ARRAY[1..2] OF BOOL;
		AX_ErrorID					: ARRAY[1..2] OF UDINT;

	MesDataExd		AT %Q*	: INV_Huawei ; 
	
	// M_INIT //
		bInit						: BOOL;


	// M_CP

		
	// M_STATEMANAGER//
	
